FUNCTION "Szukaj_Zmiany" : VOID	// FC 5
//Funkcja wykrywa zmiane w obszarze wejscie i zapamietuje. Umozliwia to wykrycie 
//zmiany stanu kazdego czujnika lini. Funkcja ograniczona jest do dlugosci 32 
//bitow.
//
//Wersja 1.0
//Rozszerzenie dzia³ania funcji do 8 bajtow
AUTHOR : Kng
NAME : Help_FC
VERSION : 0.1
VAR_INPUT
  DWORD_IN_NEW : DWORD ;
END_VAR
VAR_IN_OUT
  DWORD_IN_OLD : DWORD ;
  CHANGE : BOOL ;
END_VAR
VAR_TEMP
  DWORD_TEST : DWORD ;
  Temp_Bit_1 : BOOL ;
  Temp_Bit_2 : BOOL ;
END_VAR
BEGIN
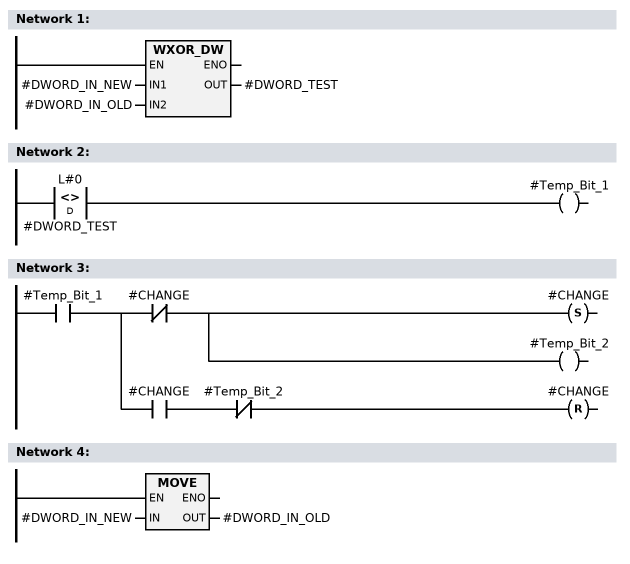
NETWORK
TITLE =
//Sprawdz czy nastapila zmiana
      L     #DWORD_IN_NEW;
      L     #DWORD_IN_OLD;
      XOD;
      T     #DWORD_TEST;
NETWORK
TITLE =
////wykrycie zmiany stanu 
      L     L#0;
      L     #DWORD_TEST;
      <>D;
      =     #Temp_Bit_1;
NETWORK
TITLE =
//Zapisz wykryta zminane
      A     #Temp_Bit_1;
      =     L 5.0;
      A     L 5.0;
      AN    #CHANGE;
      S     #CHANGE;
      =     #Temp_Bit_2;
      A     L 5.0;
      A     #CHANGE;
      AN    #Temp_Bit_2;
      R     #CHANGE;
NETWORK
TITLE =
//Przypisz wartosc obecna jako stara
      L     #DWORD_IN_NEW;
      T     #DWORD_IN_OLD;
END_FUNCTION

FUNCTION "FC_Lampki" : VOID	// FC 6
VERSION : 0.1
VAR_INPUT
  in_0 : BOOL ;
  in_1 : BOOL ;
  in_2 : BOOL ;
  in_3 : BOOL ;
  in_4 : BOOL ;
  in_5 : BOOL ;
  in_6 : BOOL ;
  in_7 : BOOL ;
  Test : BOOL ;
END_VAR
VAR_OUTPUT
  out_0 : BOOL ;
  out_1 : BOOL ;
  out_2 : BOOL ;
  out_3 : BOOL ;
  out_4 : BOOL ;
  out_5 : BOOL ;
  out_6 : BOOL ;
  out_7 : BOOL ;
END_VAR
BEGIN
NETWORK
TITLE =
//przyporzadkowanie wejsc do wyjs
//0
      O     #in_0;
      O     #Test;
      =     #out_0;
//1
      O     #in_1;
      O     #Test;
      =     #out_1;
//2
      O     #in_2;
      O     #Test;
      =     #out_2;
//3
      O     #in_3;
      O     #Test;
      =     #out_3;
//4
      O     #in_4;
      O     #Test;
      =     #out_4;
//5
      O     #in_5;
      O     #Test;
      =     #out_5;
//6
      O     #in_6;
      O     #Test;
      =     #out_6;
//7
      O     #in_7;
      O     #Test;
      =     #out_7;
END_FUNCTION

FUNCTION "Szukaj_Zmiany_2" : VOID	// FC 7
//Funkcja wykrywa zmiane w obszarze wejscie i zapamietuje. Umozliwia to wykrycie 
//zmiany stanu kazdego czujnika lini. Funkcja ograniczona jest do dlugosci 32 
//bitow.
//
//Wersja 1.0
//Rozszerzenie dzia³ania funcji do 8 bajtow
AUTHOR : Kng
NAME : Help_FC
VERSION : 0.1
VAR_INPUT
  DWORD_IN_NEW : DWORD ;
END_VAR
VAR_OUTPUT
  CHANGE : BOOL ;
END_VAR
VAR_IN_OUT
  DWORD_IN_OLD : DWORD ;
END_VAR
BEGIN
NETWORK
TITLE =
//Sprawdz czy nastapila zmiana
      L     #DWORD_IN_NEW;
      L     #DWORD_IN_OLD;
      XOD;
      L     L#0;
      <>D;
      =     #CHANGE;
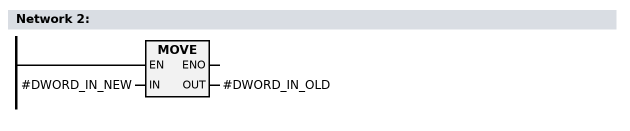
NETWORK
TITLE =
//Przypisz wartosc obecna jako stara
      L     #DWORD_IN_NEW;
      T     #DWORD_IN_OLD;
END_FUNCTION

FUNCTION "Toggle" : VOID	// FC 8
//Funcja zmienia stan wyjscia gdy ktore kolwiek wejscie zostanie wyzwolone
AUTHOR : Kng
NAME : Help_FC
VERSION : 0.1
VAR_INPUT
  Wyzwolenie_1 : BOOL ;
  Wyzwolenie_2 : BOOL ;
  Wyzwolenie_3 : BOOL ;
  Wyzwolenie_4 : BOOL ;
END_VAR
VAR_IN_OUT
  TOGGLE : BOOL ;
END_VAR
VAR_TEMP
  Temp_Bit_2 : BOOL ;
END_VAR
BEGIN
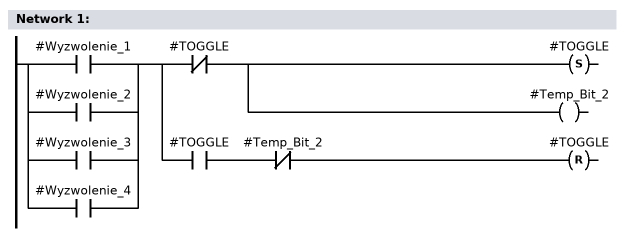
NETWORK
TITLE =
//Zapisz wykryta zminane
      O     #Wyzwolenie_1;
      O     #Wyzwolenie_2;
      O     #Wyzwolenie_3;
      O     #Wyzwolenie_4;
      =     L 1.0;
      A     L 1.0;
      AN    #TOGGLE;
      S     #TOGGLE;
      =     #Temp_Bit_2;
      A     L 1.0;
      A     #TOGGLE;
      AN    #Temp_Bit_2;
      R     #TOGGLE;
END_FUNCTION

FUNCTION "Sterwanie_Swiatlo" : VOID	// FC 9
VERSION : 0.1
VAR_TEMP
  Help_Bit : BOOL ;
END_VAR
BEGIN
NETWORK
TITLE =
//Ten Network celowo jest wolny
NETWORK
TITLE =
//Wyszczegolnienie bledow
//Not AUS Adres 27 (szafa)
//Kod :0001
      A     "Not_Aus_27_OK";
      L     B#16#1;
      JCN   KOD;
//Not AUS Adres 28 (poczatek lini)
//Kod :0010
      A     "Not_Aus_28_OK";
      L     B#16#2;
      JCN   KOD;
//Not AUS Adres 29 (srodek lini)
//Kod :0011
      A     "Not_Aus_29_OK";
      L     B#16#3;
      JCN   KOD;
//Not AUS Adres 30 (koniec lini)
//Kod :0100
      A     "Not_Aus_30_OK";
      L     B#16#4;
      JCN   KOD;
//Sprawdzenie bezpiecznikow w szafie
//Kod:0101
      A     "Fuse_OK";
      L     B#16#5;
      JCN   KOD;
//Sprwadzenie przekaznika bezpieczenstwa
//Kod:0110
      A     "Przekaznik_Bezp_OK";
      L     B#16#6;
      JCN   KOD;
//Sprawdzenie Falownikow Lini    
//Kod:0111
      A     "Falowniki_OK";
      L     B#16#7;
      JCN   KOD;
//Not AUS Adres 31 (koniec lini)
//Kod :1000
      A     "Not_Aus_31_OK";
      L     B#16#8;
      JCN   KOD;
//Sprawdzenie czy jest wlaczony  stop
//Kod:1111
      AN    "Marka_Start_Stop";
      L     B#16#F;
      JCN   KOD;
//Not AUS Adres (Strefa Bindownica)
//Kod :1001
      A     "Strefa_Bind_Zamk";
      L     B#16#9;
      JCN   KOD;
//Not AUS Adres (Strefa Bindownica)
//Kod :1010
      A     "Przek_Rejonu_Bind_Ok";
      L     B#16#10;
      JCN   KOD;
//Brak bledu maszyna pracuje
//Kod:0000
      L     B#16#0;
//Przekaz kod bledu
KOD:  T     "Byte_Bledu";
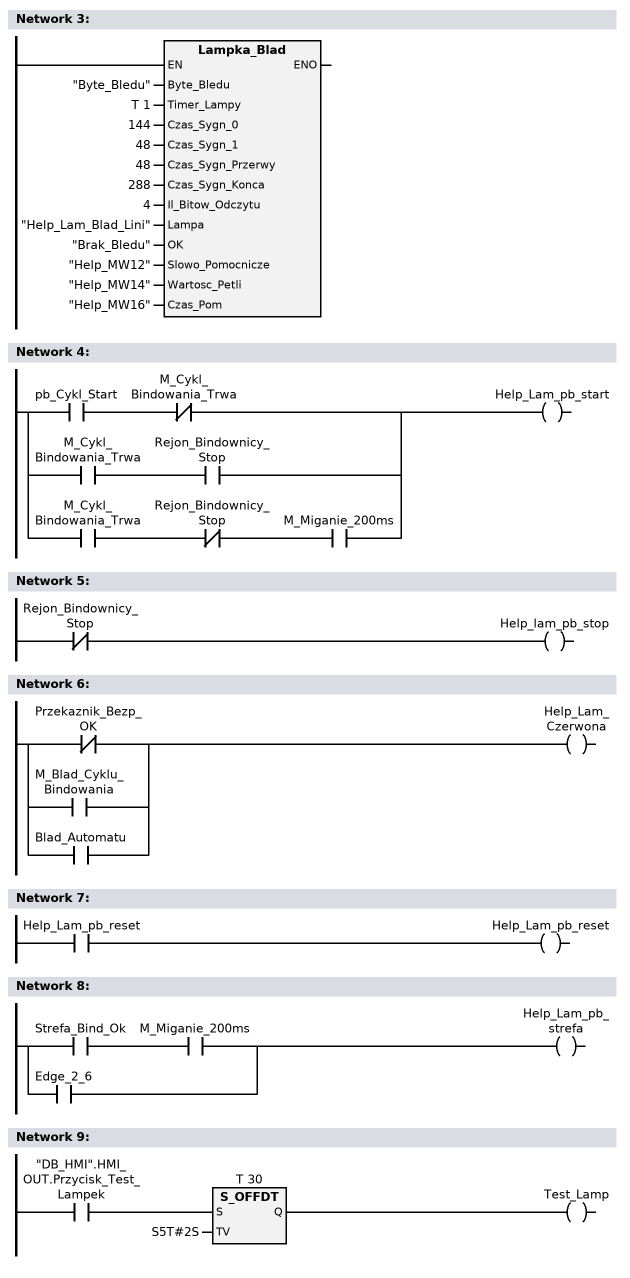
NETWORK
TITLE =
//Lampka bledu
      CALL  "Lampka_Blad" (
           Byte_Bledu               := "Byte_Bledu",
           Timer_Lampy              := T 1,
           Czas_Sygn_0              := 144,
           Czas_Sygn_1              := 48,
           Czas_Sygn_Przerwy        := 48,
           Czas_Sygn_Konca          := 288,
           Il_Bitow_Odczytu         := 4,
           Lampa                    := "Help_Lam_Blad_Lini",
           OK                       := "Brak_Bledu",
           Slowo_Pomocnicze         := "Help_MW12",
           Wartosc_Petli            := "Help_MW14",
           Czas_Pom                 := "Help_MW16");
NETWORK
TITLE =
//Lampka pb start
      A     "pb_Cykl_Start";
      AN    "M_Cykl_Bindowania_Trwa";
      O;
      A     "M_Cykl_Bindowania_Trwa";
      A     "Rejon_Bindownicy_Stop";
      O;
      A     "M_Cykl_Bindowania_Trwa";
      AN    "Rejon_Bindownicy_Stop";
      A     "M_Miganie_200ms";
      =     "Help_Lam_pb_start";
NETWORK
TITLE =
//Lampka stop
      AN    "Rejon_Bindownicy_Stop";
      =     "Help_lam_pb_stop";
NETWORK
TITLE =
      ON    "Przekaznik_Bezp_OK";
      O     "M_Blad_Cyklu_Bindowania";
      O     "Blad_Automatu";
      =     "Help_Lam_Czerwona";
NETWORK
TITLE =
//Miga reset
      A     "Help_Lam_pb_reset";
      =     "Help_Lam_pb_reset";
NETWORK
TITLE =
//Lampka bezpieczenstwa strefa
      A     "Strefa_Bind_Ok";
      A     "M_Miganie_200ms";
      O     "Edge_2_6";
      =     "Help_Lam_pb_strefa";
NETWORK
TITLE =
//Test Lampek z timmerem przedluzonym
      A     "DB_HMI".HMI_OUT.Przycisk_Test_Lampek;
      L     S5T#2S;
      SF    T 30;
      NOP   0;
      NOP   0;
      NOP   0;
      A     T 30;
      =     "Test_Lamp";
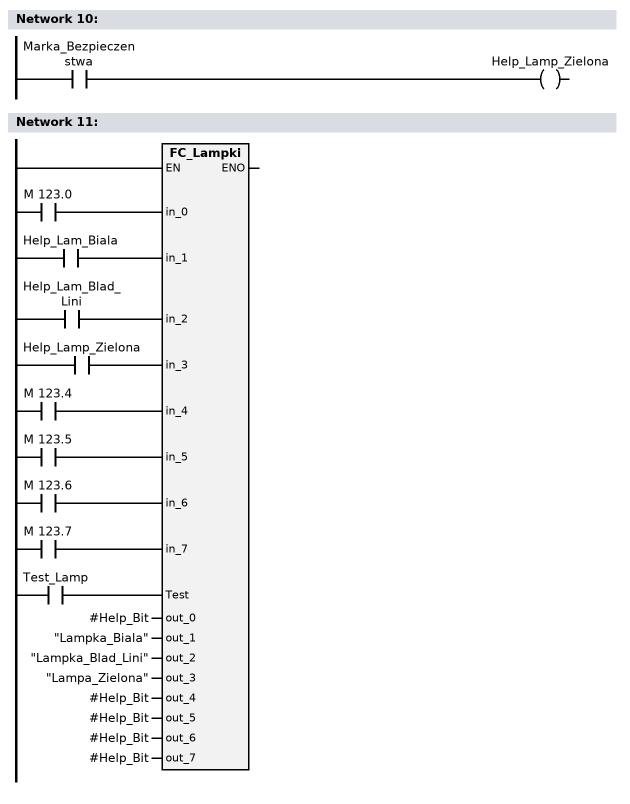
NETWORK
TITLE =
//linia pracuje
      A     "Marka_Bezpieczenstwa";
      =     "Help_Lamp_Zielona";
NETWORK
TITLE =
//Lampki na szafie sterowniczej sa troche przesuniete bo brakuje zielonej
      A     M 123.0;
      =     L 1.0;
      BLD   103;
      A     "Help_Lam_Biala";
      =     L 1.1;
      BLD   103;
      A     "Help_Lam_Blad_Lini";
      =     L 1.2;
      BLD   103;
      A     "Help_Lamp_Zielona";
      =     L 1.3;
      BLD   103;
      A     M 123.4;
      =     L 1.4;
      BLD   103;
      A     M 123.5;
      =     L 1.5;
      BLD   103;
      A     M 123.6;
      =     L 1.6;
      BLD   103;
      A     M 123.7;
      =     L 1.7;
      BLD   103;
      A     "Test_Lamp";
      =     L 2.0;
      BLD   103;
      CALL  "FC_Lampki" (
           in_0                     := L 1.0,
           in_1                     := L 1.1,
           in_2                     := L 1.2,
           in_3                     := L 1.3,
           in_4                     := L 1.4,
           in_5                     := L 1.5,
           in_6                     := L 1.6,
           in_7                     := L 1.7,
           Test                     := L 2.0,
           out_0                    := #Help_Bit,
           out_1                    := "Lampka_Biala",
           out_2                    := "Lampka_Blad_Lini",
           out_3                    := "Lampa_Zielona",
           out_4                    := #Help_Bit,
           out_5                    := #Help_Bit,
           out_6                    := #Help_Bit,
           out_7                    := #Help_Bit);
      NOP   0;
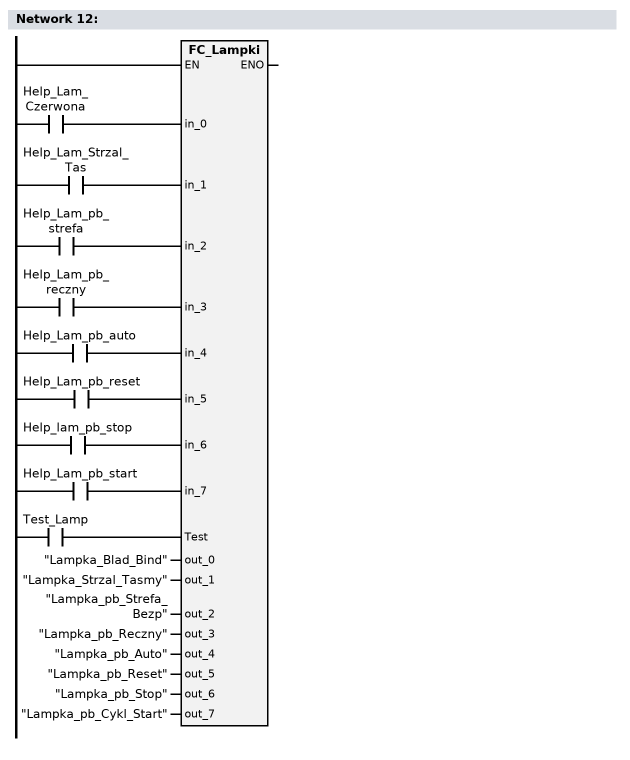
NETWORK
TITLE =
//funkcja zarzadzajaca lampami
//Lampki na panelu operatorskim
      A     "Help_Lam_Czerwona";
      =     L 1.0;
      BLD   103;
      A     "Help_Lam_Strzal_Tas";
      =     L 1.1;
      BLD   103;
      A     "Help_Lam_pb_strefa";
      =     L 1.2;
      BLD   103;
      A     "Help_Lam_pb_reczny";
      =     L 1.3;
      BLD   103;
      A     "Help_Lam_pb_auto";
      =     L 1.4;
      BLD   103;
      A     "Help_Lam_pb_reset";
      =     L 1.5;
      BLD   103;
      A     "Help_lam_pb_stop";
      =     L 1.6;
      BLD   103;
      A     "Help_Lam_pb_start";
      =     L 1.7;
      BLD   103;
      A     "Test_Lamp";
      =     L 2.0;
      BLD   103;
      CALL  "FC_Lampki" (
           in_0                     := L 1.0,
           in_1                     := L 1.1,
           in_2                     := L 1.2,
           in_3                     := L 1.3,
           in_4                     := L 1.4,
           in_5                     := L 1.5,
           in_6                     := L 1.6,
           in_7                     := L 1.7,
           Test                     := L 2.0,
           out_0                    := "Lampka_Blad_Bind",
           out_1                    := "Lampka_Strzal_Tasmy",
           out_2                    := "Lampka_pb_Strefa_Bezp",
           out_3                    := "Lampka_pb_Reczny",
           out_4                    := "Lampka_pb_Auto",
           out_5                    := "Lampka_pb_Reset",
           out_6                    := "Lampka_pb_Stop",
           out_7                    := "Lampka_pb_Cykl_Start");
      NOP   0;
END_FUNCTION

FUNCTION "Lampka_Blad" : VOID	// FC 10
//Funkcja odowiada za generowanie kodu bledu w postaci sekwencji impulsow 
//swietlnych. Maksymalna ilosc imulsow kodu wynosi 8(dl. jednego bajtu).
//Przyukladowa sekwencja kodu to 0001 (sygnal: krotki,krotki,krotki,dlugi).
//
//Kod braku bledu to 0000-przy ustawionej liczbie bitow odczytywanych na 4
//
AUTHOR : Kng
NAME : Error
VERSION : 0.1
VAR_INPUT
  Byte_Bledu : BYTE ;	//Byte wejsciowy kodu bledu
  Timer_Lampy : TIMER ;
  Czas_Sygn_0 : S5TIME ;	//Czas sygnalu dla zera
  Czas_Sygn_1 : S5TIME ;	//Czas sygnalu dla jeden
  Czas_Sygn_Przerwy : S5TIME ;	//Czas sygnalu przerwy pomiedzy impulsami
  Czas_Sygn_Konca : S5TIME ;	//Czas sygnalu konca sekwencji bledu
  Il_Bitow_Odczytu : INT ;	//Ilosc bitow odczytu sekwencji
END_VAR
VAR_OUTPUT
  Lampa : BOOL ;	//Wyjscie sterujace lampa
  OK : BOOL ;	//Brak bledow kod:0000
END_VAR
VAR_IN_OUT
  Slowo_Pomocnicze : WORD ;	//Slowo pomocnicze
  Wartosc_Petli : INT ;	//Wartosc petli
  Czas_Pom : S5TIME ;
END_VAR
VAR_TEMP
  Help_Edge_1 : BOOL ;
  Help_Edge_2 : BOOL ;
  Help_Edge_3 : BOOL ;
  Help_Edge_4 : BOOL ;
  Help_Edge_5 : BOOL ;
  Help_Lampa : BOOL ;
  Help_Timer_Gora : BOOL ;
  Help_Przerwa : BOOL ;
  Help_Timer_Dol : BOOL ;
  Help_Sek_Kon : BOOL ;
  Help_Timer_Kon : BOOL ;
  Help_Powrot : BOOL ;
  Help_Bit_Stop : BOOL ;
  Help_Bit_1_5 : BOOL ;
  Help_Bit_1_6 : BOOL ;
  Help_Bit_1_7 : BOOL ;
  Help_Word_2 : WORD ;
END_VAR
BEGIN
NETWORK
TITLE =
//Funkcja nie wykrywa bledu gdy transmisja 0000
      L     #Byte_Bledu;
      L     0;
      ==I;
      R     #Help_Bit_Stop;
      JC    good;
      L     #Byte_Bledu;
      L     B#16#F;
      ==I;
      JC    stop;
// Odczytanie zmiennych pomocniczych
      L     #Slowo_Pomocnicze;
      T     LW 0;
//Wyznaczenie sekwencji bledu
NETWORK
TITLE =
      O     #Help_Timer_Gora;
      O     #Help_Timer_Dol;
      O     #Help_Timer_Kon;
      JC    play;
// Sekwencja konca
      A     #Help_Sek_Kon;
      JCN   et_4;
      SET;
      S     #Help_Timer_Kon;
      L     #Czas_Sygn_Konca;
      T     #Czas_Pom;
      JU    play;
et_4: NOP   0;
//Sekwencja przerwy
      A     #Help_Przerwa;
      JCN   et_1;
      SET;
      S     #Help_Timer_Dol;
      L     #Czas_Sygn_Przerwy;
      T     #Czas_Pom;
      JU    play;
et_1: NOP   0;
//Wyznaczenie sekwencji bledu
//     L     #Il_Bitow_Odczytu           //skres to by uzyskac czytanie w druga
      L     #Wartosc_Petli;
      L     1;
      -I;
      L     #Byte_Bledu;
      SRW;
      T     #Help_Word_2;
//Zabranie bitu sekwencji
      A     L 3.0;	//bit po przesunieciu o odpowiednia sekwencje
      JCN   et_0;
//Czas sygnalu krotkiego
      SET;
      =     #Help_Timer_Gora;
      L     #Czas_Sygn_1;
      T     #Czas_Pom;
      JU    play;
et_0: NOP   0;
//Czas sygnalu dlugiego
      SET;
      =     #Help_Timer_Gora;
      L     #Czas_Sygn_0;
      T     #Czas_Pom;
      JU    play;
//Puszczenie sygnalu timer'a
//***************************************************************
play: O     #Help_Timer_Gora;
      O     #Help_Timer_Dol;
      O     #Help_Timer_Kon;
      AN    #Help_Powrot;
      L     #Czas_Pom;
      SE    #Timer_Lampy;
      A     #Timer_Lampy;
      =     #Help_Lampa;
//***************************************************************
//Przejscie do przerwy
      A     #Help_Timer_Gora;
      A     #Help_Lampa;
      FN    #Help_Edge_2;
      S     #Help_Przerwa;
      R     #Help_Edge_2;
      R     #Help_Timer_Gora;
      JC    play;
//Reset przerwy
      A     #Help_Timer_Dol;
      A     #Help_Lampa;
      FN    #Help_Edge_3;
      R     #Help_Przerwa;
      R     #Help_Edge_3;
      R     #Help_Timer_Dol;
      JC    play;
//Uruchomienie timer'a konca sekwencji
      A     #Help_Timer_Kon;
      A     #Help_Lampa;
      FN    #Help_Edge_5;
      R     #Help_Sek_Kon;
      R     #Help_Timer_Kon;
      R     #Help_Edge_5;
      JC    play;
//Dekrementacja licznika przesuniec bitow
      A     #Help_Przerwa;
      FP    #Help_Edge_4;
      JCN   et_2;
      L     #Wartosc_Petli;
      L     1;
      -I;
      T     #Wartosc_Petli;
et_2: NOP   0;
//Sekwencja konczaca
      L     #Wartosc_Petli;
      L     0;
      <=I;
      JCN   et_3;
      SET;
      S     #Help_Sek_Kon;
      L     #Il_Bitow_Odczytu;
      T     #Wartosc_Petli;
et_3: NOP   0;
NETWORK
TITLE =
//Wystawienie wyjsc
      A     #Help_Timer_Gora;
      A     #Help_Lampa;
      AN    #Help_Timer_Dol;
      AN    #Help_Timer_Kon;
      =     #Lampa;
NETWORK
TITLE =
      SET;
      R     #Help_Powrot;
      R     #OK;
      L     LW 0;
      T     #Slowo_Pomocnicze;
      BEU;
NETWORK
TITLE =
stop: NOP   0;
      SET;
      S     #Help_Bit_Stop;
good: NOP   0;
      A     #Help_Bit_Stop;
      =     #Lampa;
//wyzeruj wartosci pomocnicze
      L     0;
      T     LW 0;
//Przypisz ilosc petli by zaczynac od pelnego bledu
      L     #Il_Bitow_Odczytu;
      T     #Wartosc_Petli;
//Wylaczenie swiecenie lampy  i umozliwienie powrotu do pracujacego timera
      SET;
      R     #Help_Bit_Stop;
      R     #Timer_Lampy;
      S     #Help_Powrot;
      S     #OK;
      L     LW 0;
      T     #Slowo_Pomocnicze;
END_FUNCTION

FUNCTION "Przyporzadkowanie_Wejsc" : VOID	// FC 20
//Pobranie z bloku db stanu wejsc sieci asi i przyporzadkowanie do odpowiedniego 
//urzadzenia lini.
//NW35-adresy B
//
//
//Opis sygnalow od bindownicy:
//banda 23, 24, 1, 2 tworza zestaw tasm maszyny bindujacej
//obr 15 to obrotnica bindownicy
//25,26- to kurtyny
//16-rygiel
//17-modul resetu
AUTHOR : Kng
NAME : Help_FC
VERSION : 0.1
VAR_TEMP
  Help_Bit_1 : BOOL ;
  Help_Bit_2 : BOOL ;
  Help_Word_1 : INT ;
  Help_Word_2 : INT ;
END_VAR
BEGIN
NETWORK
TITLE =
//Ten network celowo jest wolny
NETWORK
TITLE =
NETWORK
TITLE = Silnik ok
//Banda Adres 1
      A     "Asi_input".Adres_1_bit_0;
      O     "Zawsze_True";	//dodane
      =     "AIO".Banda_1.Silnik_OK;
      A     "Asi_input".Adres_1_bit_1;
      =     "AIO".Banda_1.Rezerwa_Silnik;
      A     "Asi_input".Adres_1_bit_2;
      =     "AIO".Banda_1.Foto_1;
      A     "Asi_input".Adres_1_bit_3;
      =     "AIO".Banda_1.Foto_2;
NETWORK
TITLE = Silnik ok
//Banda Adres 2
      A     "Asi_input".Adres_2_bit_0;
      O     "Zawsze_True";
      =     "AIO".Banda_2.Silnik_OK;
      A     "Asi_input".Adres_2_bit_1;
      =     "AIO".Banda_2.Rezerwa_Silnik;
      A     "Asi_input".Adres_2_bit_2;
      =     "AIO".Banda_2.Foto_1;
      A     "Asi_input".Adres_2_bit_3;
      =     "AIO".Banda_2.Foto_2;
NETWORK
TITLE = Silnik ok
//Banda Adres 3
      A     "Asi_input".Adres_3_bit_0;
      =     "AIO".Banda_3.Silnik_OK;
      A     "Asi_input".Adres_3_bit_1;
      =     "AIO".Banda_3.Rezerwa_Silnik;
      A     "Asi_input".Adres_3_bit_2;
      =     "AIO".Banda_3.Foto_1;
      A     "Asi_input".Adres_3_bit_3;
      =     "AIO".Banda_3.Foto_2;
NETWORK
TITLE = Silnik ok
//Banda Adres 4
      A     "Asi_input".Adres_4_bit_0;
      =     "AIO".Banda_4.Silnik_OK;
      A     "Asi_input".Adres_4_bit_1;
      =     "AIO".Banda_4.Rezerwa_Silnik;
      A     "Asi_input".Adres_4_bit_2;
      =     "AIO".Banda_4.Foto_1;
      A     "Asi_input".Adres_4_bit_3;
      =     "AIO".Banda_4.Foto_2;
NETWORK
TITLE = Silnik ok
//Banda Adres 5
      A     "Asi_input".Adres_5_bit_0;
      =     "AIO".Banda_5.Silnik_OK;
      A     "Asi_input".Adres_5_bit_1;
      =     "AIO".Banda_5.Rezerwa_Silnik;
      A     "Asi_input".Adres_5_bit_2;
      =     "AIO".Banda_5.Foto_1;
      A     "Asi_input".Adres_5_bit_3;
      =     "AIO".Banda_5.Foto_2;
NETWORK
TITLE = Silnik ok
//Banda Adres 6
      A     "Asi_input".Adres_6_bit_0;
      =     "AIO".Banda_6.Silnik_OK;
      A     "Asi_input".Adres_6_bit_1;
      =     "AIO".Banda_6.Rezerwa_Silnik;
      A     "Asi_input".Adres_6_bit_2;
      =     "AIO".Banda_6.Foto_1;
      A     "Asi_input".Adres_6_bit_3;
      =     "AIO".Banda_6.Foto_2;
NETWORK
TITLE = Silnik ok
//Banda Adres 7
      A     "Asi_input".Adres_7_bit_0;
      =     "AIO".Banda_7.Silnik_OK;
      A     "Asi_input".Adres_7_bit_1;
      =     "AIO".Banda_7.Rezerwa_Silnik;
      A     "Asi_input".Adres_7_bit_2;
      =     "AIO".Banda_7.Foto_1;
      A     "Asi_input".Adres_7_bit_3;
      =     "AIO".Banda_7.Foto_2;
NETWORK
TITLE = Silnik ok
//Banda Adres 8
      A     "Asi_input".Adres_8_bit_0;
      =     "AIO".Banda_8.Silnik_OK;
      A     "Asi_input".Adres_8_bit_1;
      =     "AIO".Banda_8.Rezerwa_Silnik;
      A     "Asi_input".Adres_8_bit_2;
      =     "AIO".Banda_8.Foto_1;
      A     "Asi_input".Adres_8_bit_3;
      =     "AIO".Banda_8.Foto_2;
NETWORK
TITLE = Silnik ok
//Banda Adres 9
      A     "Asi_input".Adres_9_bit_0;
      =     "AIO".Banda_9.Silnik_OK;
      A     "Asi_input".Adres_9_bit_1;
      =     "AIO".Banda_9.Rezerwa_Silnik;
      A     "Asi_input".Adres_9_bit_2;
      =     "AIO".Banda_9.Foto_1;
      A     "Asi_input".Adres_9_bit_3;
      =     "AIO".Banda_9.Foto_2;
//Info do foliarki o zajetosci lini
      A     "AIO".Banda_9.Foto_1;
      =     "MPI_GD".OUT.Foto_Banda_9;
//-
NETWORK
TITLE = Silnik ok
//Banda Adres 10.Banda nalezy do foliarki.
      A     "Asi_input".Adres_10_bit_0;
      =     "AIO".Banda_10.Silnik_OK;
      A     "Asi_input".Adres_10_bit_1;
      =     "AIO".Banda_10.Rezerwa_Silnik;
      A     "Asi_input".Adres_10_bit_2;
      =     "AIO".Banda_10.Foto_1;
      A     "Asi_input".Adres_10_bit_3;
      =     "AIO".Banda_10.Foto_2;
//Sygnaly do foliarki
      A     "AIO".Banda_10.Silnik_OK;
      =     "MPI_GD".OUT.Silnik_10_OK;
//-
      A     "AIO".Banda_10.Foto_1;
      =     "MPI_GD".OUT.Foto_1_Banda_10;
//-
      A     "AIO".Banda_10.Foto_2;
      =     "MPI_GD".OUT.Foto_2_Banda_10;
NETWORK
TITLE = Silnik ok
//Banda Adres 11. Banda nalezy do foliarki.
      A     "Asi_input".Adres_11_bit_0;
      =     "AIO".Banda_11.Silnik_OK;
      A     "Asi_input".Adres_11_bit_1;
      =     "AIO".Banda_11.Rezerwa_Silnik;
      A     "Asi_input".Adres_11_bit_2;
      =     "AIO".Banda_11.Foto_1;
      A     "Asi_input".Adres_11_bit_3;
      =     "AIO".Banda_11.Foto_2;
//Sygnaly do foliarki
      A     "AIO".Banda_11.Silnik_OK;
      =     "MPI_GD".OUT.Silnik_11_OK;
//-
      A     "AIO".Banda_11.Foto_1;
      =     "MPI_GD".OUT.Foto_Banda_11;
NETWORK
TITLE = Silnik ok
//Banda Adres 12
      A     "Asi_input".Adres_12_bit_0;
      =     "AIO".Banda_12.Silnik_OK;
      A     "Asi_input".Adres_12_bit_1;
      =     "AIO".Banda_12.Rezerwa_Silnik;
      A     "Asi_input".Adres_12_bit_2;
      =     "AIO".Banda_12.Foto_1;
      A     "Asi_input".Adres_12_bit_3;
      =     "AIO".Banda_12.Foto_2;
NETWORK
TITLE = Silnik ok
//Banda Adres 13
      A     "Asi_input".Adres_13_bit_0;
      =     "AIO".Banda_13.Silnik_OK;
      A     "Asi_input".Adres_13_bit_1;
      =     "AIO".Banda_13.Rezerwa_Silnik;
      A     "Asi_input".Adres_13_bit_2;
      =     "AIO".Banda_13.Foto_1;
      A     "Asi_input".Adres_13_bit_3;
      =     "AIO".Banda_13.Foto_2;
NETWORK
TITLE = Silnik ok
//Banda Adres 14
      A     "Asi_input".Adres_14_bit_0;
      =     "AIO".Banda_14.Silnik_OK;
      A     "Asi_input".Adres_14_bit_1;
      =     "AIO".Banda_14.Rezerwa_Silnik;
      A     "Asi_input".Adres_14_bit_2;
      =     "AIO".Banda_14.Foto_1;
      A     "Asi_input".Adres_14_bit_3;
      =     "AIO".Banda_14.Foto_2;
NETWORK
TITLE = Silnik ok
//Obrotnica Adres 15
      A     "Asi_input".Adres_15_bit_0;
      =     "AIO".Obr_15.Silnik_OK;
      A     "Asi_input".Adres_15_bit_1;
      =     "AIO".Obr_15.Rezerwa_Silnik;
      A     "Asi_input".Adres_15_bit_2;
      =     "AIO".Obr_15.Foto_1;
      A     "Asi_input".Adres_15_bit_3;
      =     "AIO".Obr_15.Foto_2;
NETWORK
TITLE = Silnik ok
//Uwaga modul safety !!!
//Rygiel Adres 16
      A     "Asi_input".Adres_16_bit_0;
      =     "AIO".Rygiel_16.OSSD_Tor_1_1;
      A     "Asi_input".Adres_16_bit_1;
      =     "AIO".Rygiel_16.OSSD_Tor_1_2;
      A     "Asi_input".Adres_16_bit_2;
      =     "AIO".Rygiel_16.OSSD_Tor_2_1;
      A     "Asi_input".Adres_16_bit_3;
      =     "AIO".Rygiel_16.OSSD_Tor_2_2;
NETWORK
TITLE = Silnik ok
//Reset kurtyn bezpieczenswa Adres 17
//Nie wykorzystywane wejscia
NETWORK
TITLE = Silnik ok
//Obrotnica Adres_18
      A     "Asi_input".Adres_18_bit_0;
      =     "AIO".Obr_18.Silnik_OK;
      A     "Asi_input".Adres_18_bit_1;
      =     "AIO".Obr_18.Rezerwa_Silnik;
      A     "Asi_input".Adres_18_bit_2;
      =     "AIO".Obr_18.Foto_1;
      A     "Asi_input".Adres_18_bit_3;
      =     "AIO".Obr_18.Foto_2;
NETWORK
TITLE = Silnik ok
//Czujniki obrotnicy 1 Adres 19
      A     "Asi_input".Adres_19_bit_0;
      =     "AIO".Czuj_19.Czujnik_0_St;
      A     "Asi_input".Adres_19_bit_1;
      =     "AIO".Czuj_19.Czujnik_Ham_0_St;
      A     "Asi_input".Adres_19_bit_2;
      =     "AIO".Czuj_19.Czujnik_Ham_90_St;
      A     "Asi_input".Adres_19_bit_3;
      =     "AIO".Czuj_19.Czujnik_90_St;
NETWORK
TITLE = Silnik ok
//Obrotnica Adres 20
      A     "Asi_input".Adres_20_bit_0;
      =     "AIO".Obr_20.Silnik_OK;
      A     "Asi_input".Adres_20_bit_1;
      =     "AIO".Obr_20.Rezerwa_Silnik;
      A     "Asi_input".Adres_20_bit_2;
      =     "AIO".Obr_20.Foto_1;
      A     "Asi_input".Adres_20_bit_3;
      =     "AIO".Obr_20.Foto_2;
NETWORK
TITLE = Silnik ok
//Czujniki Obrotnicy 2 Adres 21
      A     "Asi_input".Adres_21_bit_0;
      =     "AIO".Czuj_21.Czujnik_0_St;
      A     "Asi_input".Adres_21_bit_1;
      =     "AIO".Czuj_21.Czujnik_Ham_0_St;
      A     "Asi_input".Adres_21_bit_2;
      =     "AIO".Czuj_21.Czujnik_Ham_90_St;
      A     "Asi_input".Adres_21_bit_3;
      =     "AIO".Czuj_21.Czujnik_90_St;
NETWORK
TITLE = Silnik ok
//Czujniki Obrotnicy 2 Adres 22
      A     "Asi_input".Adres_22_bit_0;
      =     "AIO".Czuj_22.Czujnik_45_St_CW;
      A     "Asi_input".Adres_22_bit_1;
      =     "AIO".Czuj_22.Czujnik_45_St_CCW;
      A     "Asi_input".Adres_22_bit_2;
      =     "AIO".Czuj_22.Rez_0_2;
      A     "Asi_input".Adres_22_bit_3;
      =     "AIO".Czuj_22.Rez_0_3;
NETWORK
TITLE = Wejscie SEW 1
//Banda 23 znajdujaca sie bedaca banda wjazdowa do bindownicy
      A     "Asi_input".Adres_23_bit_0;
      =     "AIO".Banda_23.Silnik_OK;
      A     "Asi_input".Adres_23_bit_1;
      =     "AIO".Banda_23.Rezerwa_Silnik;
      A     "Asi_input".Adres_23_bit_2;
      =     "AIO".Banda_23.Foto_1;
      A     "Asi_input".Adres_23_bit_3;
      =     "AIO".Banda_23.Foto_2;
NETWORK
TITLE = Silnik ok
//Banda 24
      A     "Asi_input".Adres_24_bit_0;
      =     "AIO".Banda_24.Silnik_OK;
      A     "Asi_input".Adres_24_bit_1;
      =     "AIO".Banda_24.Rezerwa_Silnik;
      A     "Asi_input".Adres_24_bit_2;
      =     "AIO".Banda_24.Foto_1;
      A     "Asi_input".Adres_24_bit_3;
      =     "AIO".Banda_24.Foto_2;
NETWORK
TITLE =
//Sprawdzenie czujnikow Bezpieczenstwa lini
//Kurtyna 25
      A     "Asi_input".Adres_25_bit_0;
      =     "AIO".Kurtyna_25.OSSD_Tor_1_1;
      A     "Asi_input".Adres_25_bit_1;
      =     "AIO".Kurtyna_25.OSSD_Tor_1_2;
      A     "Asi_input".Adres_25_bit_2;
      =     "AIO".Kurtyna_25.OSSD_Tor_2_1;
      A     "Asi_input".Adres_25_bit_3;
      =     "AIO".Kurtyna_25.OSSD_Tor_2_2;
NETWORK
TITLE =
//Sprawdzenie czujnikow Bezpieczenstwa lini
//Kurtyna 26
      A     "Asi_input".Adres_26_bit_0;
      =     "AIO".Kurtyna_26.OSSD_Tor_1_1;
      A     "Asi_input".Adres_26_bit_1;
      =     "AIO".Kurtyna_26.OSSD_Tor_1_2;
      A     "Asi_input".Adres_26_bit_2;
      =     "AIO".Kurtyna_26.OSSD_Tor_2_1;
      A     "Asi_input".Adres_26_bit_3;
      =     "AIO".Kurtyna_26.OSSD_Tor_2_2;
NETWORK
TITLE = Silnik ok
//Sprawdzenie czujnikow Bezpieczenstwa lini
//Not Aus 27
      A     "Asi_input".Adres_27_bit_0;
      =     "AIO".ESTOP_27.EStop_Tor_1_1;
      A     "Asi_input".Adres_27_bit_1;
      =     "AIO".ESTOP_27.EStop_Tor_1_2;
      A     "Asi_input".Adres_27_bit_2;
      =     "AIO".ESTOP_27.EStop_Tor_2_1;
      A     "Asi_input".Adres_27_bit_3;
      =     "AIO".ESTOP_27.EStop_Tor_2_2;
NETWORK
TITLE =
//Sprawdzenie czujnikow Bezpieczenstwa lini
//Not Aus 28
      A     "Asi_input".Adres_28_bit_0;
      =     "AIO".ESTOP_28.EStop_Tor_1_1;
      A     "Asi_input".Adres_28_bit_1;
      =     "AIO".ESTOP_28.EStop_Tor_1_2;
      A     "Asi_input".Adres_28_bit_2;
      =     "AIO".ESTOP_28.EStop_Tor_2_1;
      A     "Asi_input".Adres_28_bit_3;
      =     "AIO".ESTOP_28.EStop_Tor_2_2;
NETWORK
TITLE =
//Sprawdzenie czujnikow Bezpieczenstwa lini
//Not Aus 29
      A     "Asi_input".Adres_29_bit_0;
      =     "AIO".ESTOP_29.EStop_Tor_1_1;
      A     "Asi_input".Adres_29_bit_1;
      =     "AIO".ESTOP_29.EStop_Tor_1_2;
      A     "Asi_input".Adres_29_bit_2;
      =     "AIO".ESTOP_29.EStop_Tor_2_1;
      A     "Asi_input".Adres_29_bit_3;
      =     "AIO".ESTOP_29.EStop_Tor_2_2;
NETWORK
TITLE =
//Sprawdzenie czujnikow Bezpieczenstwa lini
//Not Aus 30
      A     "Asi_input".Adres_30_bit_0;
      =     "AIO".ESTOP_30.EStop_Tor_1_1;
      A     "Asi_input".Adres_30_bit_1;
      =     "AIO".ESTOP_30.EStop_Tor_1_2;
      A     "Asi_input".Adres_30_bit_2;
      =     "AIO".ESTOP_30.EStop_Tor_2_1;
      A     "Asi_input".Adres_30_bit_3;
      =     "AIO".ESTOP_30.EStop_Tor_2_2;
NETWORK
TITLE =
//Sprawdzenie czujnikow Bezpieczenstwa lini
//Not Aus 31
      A     "Asi_input".Adres_31_bit_0;
      =     "AIO".ESTOP_31.EStop_Tor_1_1;
      A     "Asi_input".Adres_31_bit_1;
      =     "AIO".ESTOP_31.EStop_Tor_1_2;
      A     "Asi_input".Adres_31_bit_2;
      =     "AIO".ESTOP_31.EStop_Tor_2_1;
      A     "Asi_input".Adres_31_bit_3;
      =     "AIO".ESTOP_31.EStop_Tor_2_2;
NETWORK
TITLE =
//Segment adresow B
//Dotyczy jedynie bialych modulow inuput nie zawartych wyzej
NETWORK
TITLE =
//Czujnik bindownicy Adres 19B 
      A     "Asi_input".B_Adres_19_bit_0;
      =     "AIO".Czuj_19_B.Czujnik_0_St;
      A     "Asi_input".B_Adres_19_bit_1;
      =     "AIO".Czuj_19_B.Czujnik_Ham_0_St;
      A     "Asi_input".B_Adres_19_bit_2;
      =     "AIO".Czuj_19_B.Czujnik_Ham_90_St;
      A     "Asi_input".B_Adres_19_bit_3;
      =     "AIO".Czuj_19_B.Czujnik_90_St;
NETWORK
TITLE =
//Czujnik bindownicy Adres 17B 
      A     "Asi_input".B_Adres_17_bit_0;
      =     "AIO".Czuj_17_B.Czujnik_Ham_180_St;
      A     "Asi_input".B_Adres_17_bit_1;
      =     "AIO".Czuj_17_B.Czujnik_180_St;
      A     "Asi_input".B_Adres_17_bit_2;
      =     "AIO".Czuj_17_B.Czujnik_Ham_270_St;
      A     "Asi_input".B_Adres_17_bit_3;
      =     "AIO".Czuj_17_B.Czujnik_270_St;
END_FUNCTION

FUNCTION "Przyporzadkowanie_Wyjsc" : VOID	// FC 21
VERSION : 0.1
VAR_TEMP
  Temp_Word_1 : INT ;
  Help_Bit_1 : BOOL ;
END_VAR
BEGIN
NETWORK
TITLE =
//Ten Network celowo jest wolny
NETWORK
TITLE = Temporary placeholder variable
//Banda 1 Adres 1
//****************ClockWise*******************
      A     "AIO".Banda_1.CC_Wise;	//C_Wise
      =     "Asi_output".Adres_1_bit_0;
//****************CounterClockWise************
      A     "AIO".Banda_1.C_Wise;
      =     "Asi_output".Adres_1_bit_1;	//CC_Wise
//****************Wolno***********************
      A     "AIO".Banda_1.Wolno;
      O     "pb_Strefa_bezpieczenstwa";
      =     "Asi_output".Adres_1_bit_2;	//Wolno
//****************Bit_Bezpieczenstwa**********
      A     "Marka_Bezpieczenstwa";	//Safety
      =     "Asi_output".Adres_1_bit_3;
NETWORK
TITLE = Temporary placeholder variable
//Banda 2 Adres 2
//****************ClockWise*******************
      A     "AIO".Banda_2.CC_Wise;	//C_Wise
      =     "Asi_output".Adres_2_bit_0;
//****************CounterClockWise************
      A     "AIO".Banda_2.C_Wise;
      =     "Asi_output".Adres_2_bit_1;	//CC_Wise
//****************Wolno***********************
      AN    "AIO".Banda_2.Wolno;
      =     "Asi_output".Adres_2_bit_2;	//Wolno
//****************Bit_Bezpieczenstwa**********
      A     "Marka_Bezpieczenstwa";	//Safety
      =     "Asi_output".Adres_2_bit_3;
NETWORK
TITLE = Temporary placeholder variable
//Banda 3 Adres 3
//****************ClockWise*******************
      A     "Zawsze_False";	//C_Wise
      =     "Asi_output".Adres_3_bit_0;
//****************CounterClockWise************
      A     "AIO".Banda_3.C_Wise;
      =     "Asi_output".Adres_3_bit_1;	//CC_Wise
//****************Wolno***********************
      A     "Zawsze_True";
      =     "Asi_output".Adres_3_bit_2;	//Wolno
//****************Bit_Bezpieczenstwa**********
      A     "Marka_Bezpieczenstwa";	//Safety
      =     "Asi_output".Adres_3_bit_3;
NETWORK
TITLE = Temporary placeholder variable
//Banda 4 Obrotnica
//****************ClockWise*******************
      A     "AIO".Banda_4.C_Wise;	//C_Wise
      =     "Asi_output".Adres_4_bit_0;
//****************CounterClockWise************
      A     "AIO".Banda_4.CC_Wise;
      =     "Asi_output".Adres_4_bit_1;	//CC_Wise
//****************Wolno***********************
      A     "Zawsze_True";
      =     "Asi_output".Adres_4_bit_2;	//Wolno
//****************Bit_Bezpieczenstwa**********
      A     "Marka_Bezpieczenstwa";	//Safety
      =     "Asi_output".Adres_4_bit_3;
NETWORK
TITLE = Temporary placeholder variable
//Banda 5 Rolki
//****************ClockWise*******************
      A     "Zawsze_False";	//C_Wise
      =     "Asi_output".Adres_5_bit_0;
//****************CounterClockWise************
      A     "AIO".Banda_5.C_Wise;
      =     "Asi_output".Adres_5_bit_1;	//CC_Wise
//****************Wolno***********************
      A     "Zawsze_True";
      =     "Asi_output".Adres_5_bit_2;	//Wolno
//****************Bit_Bezpieczenstwa**********
      A     "Marka_Bezpieczenstwa";	//Safety
      =     "Asi_output".Adres_5_bit_3;
NETWORK
TITLE = Temporary placeholder variable
//Banda 6 Rolki
//****************ClockWise*******************
      A     "AIO".Banda_6.C_Wise;	//C_Wise
      =     "Asi_output".Adres_6_bit_0;
//****************CounterClockWise************
      A     "Zawsze_False";
      =     "Asi_output".Adres_6_bit_1;	//CC_Wise
//****************Wolno***********************
      A     "Zawsze_False";
      =     "Asi_output".Adres_6_bit_2;	//Wolno
//****************Bit_Bezpieczenstwa**********
      A     "Marka_Bezpieczenstwa";	//Safety
      =     "Asi_output".Adres_6_bit_3;
NETWORK
TITLE = Temporary placeholder variable
//Banda 7 Rolki
//****************ClockWise*******************
      A     "Zawsze_False";	//C_Wise
      =     "Asi_output".Adres_7_bit_0;
//****************CounterClockWise************
      A     "AIO".Banda_7.C_Wise;
      =     "Asi_output".Adres_7_bit_1;	//CC_Wise
//****************Wolno***********************
      A     "Zawsze_True";
      =     "Asi_output".Adres_7_bit_2;	//Wolno
//****************Bit_Bezpieczenstwa**********
      A     "Marka_Bezpieczenstwa";	//Safety
      =     "Asi_output".Adres_7_bit_3;
NETWORK
TITLE = Temporary placeholder variable
//Banda 8 Rolki
//****************ClockWise*******************
      A     "AIO".Banda_8.C_Wise;	//C_Wise
      =     "Asi_output".Adres_8_bit_0;
//****************CounterClockWise************
      A     "Zawsze_False";
      =     "Asi_output".Adres_8_bit_1;	//CC_Wise
//****************Wolno***********************
      A     "Zawsze_False";
      =     "Asi_output".Adres_8_bit_2;	//Wolno
//****************Bit_Bezpieczenstwa**********
      A     "Marka_Bezpieczenstwa";	//Safety
      =     "Asi_output".Adres_8_bit_3;
NETWORK
TITLE = Temporary placeholder variable
//Banda 9 Rolki
//****************ClockWise*******************
      A     "Zawsze_False";	//C_Wise
      =     "Asi_output".Adres_9_bit_0;
//****************CounterClockWise************
      A     "AIO".Banda_9.C_Wise;
      =     "Asi_output".Adres_9_bit_1;	//CC_Wise
//****************Wolno***********************
      A     "Zawsze_True";
      =     "Asi_output".Adres_9_bit_2;	//Wolno
//****************Bit_Bezpieczenstwa**********
      A     "Marka_Bezpieczenstwa";	//Safety
      =     "Asi_output".Adres_9_bit_3;
NETWORK
TITLE = Temporary placeholder variable
//Banda 10 Rolki
//Uwaga Banda ta nalezy do foliarki
//Sygnaly z foliarki
      A     "MPI_GD".IN.Motor_10_Lewo;
      =     "AIO".Banda_10.C_Wise;
      A     "MPI_GD".IN.Motor_10_Prawo;
      =     "AIO".Banda_10.CC_Wise;
//****************ClockWise*******************
      A     "AIO".Banda_10.C_Wise;	//C_Wise
      =     "Asi_output".Adres_10_bit_0;
//****************CounterClockWise************
      A     "AIO".Banda_10.CC_Wise;
      =     "Asi_output".Adres_10_bit_1;	//CC_Wise
//****************Wolno***********************
      A     "Zawsze_True";
      =     "Asi_output".Adres_10_bit_2;	//Wolno
//****************Bit_Bezpieczenstwa**********
      A     "Marka_Bezpieczenstwa";	//Safety
      =     "Asi_output".Adres_10_bit_3;
NETWORK
TITLE = Temporary placeholder variable
//Banda 11 Rolki
//Uwaga Banda ta nalezy do foliarki
//Sygnaly z foliarki
      A     "MPI_GD".IN.Motor_11_Lewo;
      =     "AIO".Banda_11.C_Wise;
      A     "MPI_GD".IN.Motor_11_Prawo;
      =     "AIO".Banda_11.CC_Wise;
//****************ClockWise*******************
      A     "AIO".Banda_11.C_Wise;	//C_Wise
      =     "Asi_output".Adres_11_bit_0;
//****************CounterClockWise************
      A     "AIO".Banda_11.CC_Wise;
      =     "Asi_output".Adres_11_bit_1;	//CC_Wise
//****************Wolno***********************
      A     "Zawsze_True";
      =     "Asi_output".Adres_11_bit_2;	//Wolno
//****************Bit_Bezpieczenstwa**********
      A     "Marka_Bezpieczenstwa";	//Safety
      =     "Asi_output".Adres_11_bit_3;
NETWORK
TITLE = Temporary placeholder variable
//Banda 12 Rolki wlot 2 na obrotnice
//****************ClockWise*******************
      A     "AIO".Banda_12.C_Wise;	//C_Wise
      =     "Asi_output".Adres_12_bit_0;
//****************CounterClockWise************
      A     "Zawsze_False";
      =     "Asi_output".Adres_12_bit_1;	//CC_Wise
//****************Wolno***********************
      A     "Zawsze_False";
      =     "Asi_output".Adres_12_bit_2;	//Wolno
//****************Bit_Bezpieczenstwa**********
      A     "Marka_Bezpieczenstwa";	//Safety
      =     "Asi_output".Adres_12_bit_3;
NETWORK
TITLE = Temporary placeholder variable
//Banda 13 Adres 13 Rolki na obrotnicy
//****************ClockWise*******************
      A     "AIO".Banda_13.C_Wise;	//C_Wise
      =     "Asi_output".Adres_13_bit_0;
//****************CounterClockWise************
      A     "AIO".Banda_13.CC_Wise;
      =     "Asi_output".Adres_13_bit_1;	//CC_Wise
//****************Wolno***********************
      A     "Zawsze_False";
      =     "Asi_output".Adres_13_bit_2;	//Wolno
//****************Bit_Bezpieczenstwa**********
      A     "Marka_Bezpieczenstwa";	//Safety
      =     "Asi_output".Adres_13_bit_3;
NETWORK
TITLE = Temporary placeholder variable
//Banda 14 Adres 14 Wylot z maszyny
//****************ClockWise*******************
      A     "AIO".Banda_14.C_Wise;	//C_Wise
      =     "Asi_output".Adres_14_bit_0;
//****************CounterClockWise************
      A     "Zawsze_False";
      =     "Asi_output".Adres_14_bit_1;	//CC_Wise
//****************Wolno***********************
      A     "Zawsze_False";
      =     "Asi_output".Adres_14_bit_2;	//Wolno
//****************Bit_Bezpieczenstwa**********
      A     "Marka_Bezpieczenstwa";	//Safety
      =     "Asi_output".Adres_14_bit_3;
NETWORK
TITLE = Temporary placeholder variable
//Obrotnica 15 Adres 15
//****************ClockWise*******************
      A     "AIO".Obr_15.C_Wise;
      =     "Asi_output".Adres_15_bit_0;
//****************CounterClockWise************
      A     "AIO".Obr_15.CC_Wise;
      =     "Asi_output".Adres_15_bit_1;	//CC_Wise
//****************Wolno***********************
      AN    "AIO".Obr_15.Wolno;
      =     "Asi_output".Adres_15_bit_2;	//Wolno
//****************Bit_Bezpieczenstwa**********
      A     "Marka_Bezpieczenstwa";	//Safety
      =     "Asi_output".Adres_15_bit_3;
NETWORK
TITLE =
//adres 16 rygiel brak output
NETWORK
TITLE = Temporary placeholder variable
//adres 17 reset kurtyn
//****************Reset wlot *****************
      A     "AIO".Reset_17.Reset_Wlot;
      =     "Asi_output".Adres_17_bit_0;	//reset wlot
//****************Reset wylot ****************
      A     "AIO".Reset_17.Reset_Wylot;
      =     "Asi_output".Adres_17_bit_1;	//reset wylot
NETWORK
TITLE = Temporary placeholder variable
//Obrotnica 18  Adres 18
//****************ClockWise*******************
      A     "AIO".Obr_18.C_Wise;
      =     "Asi_output".Adres_18_bit_0;
//****************CounterClockWise************
      A     "AIO".Obr_18.CC_Wise;
      =     "Asi_output".Adres_18_bit_1;	//CC_Wise
//****************Wolno***********************
      A     "AIO".Obr_18.Wolno;
      =     "Asi_output".Adres_18_bit_2;	//Wolno
//****************Bit_Bezpieczenstwa**********
      A     "Marka_Bezpieczenstwa";	//Safety
      =     "Asi_output".Adres_18_bit_3;
NETWORK
TITLE = Temporary placeholder variable
//Adres 19 brak sygnalow output
NETWORK
TITLE = Temporary placeholder variable
//Obrotnica 20 Adres 20
//****************ClockWise*******************
      A     "AIO".Obr_20.C_Wise;
      =     "Asi_output".Adres_20_bit_0;
//****************CounterClockWise************
      A     "AIO".Obr_20.CC_Wise;
      =     "Asi_output".Adres_20_bit_1;	//CC_Wise
//****************Wolno***********************
      A     "AIO".Obr_20.Wolno;
      =     "Asi_output".Adres_20_bit_2;	//Wolno
//****************Bit_Bezpieczenstwa**********
      A     "Marka_Bezpieczenstwa";	//Safety
      =     "Asi_output".Adres_20_bit_3;
NETWORK
TITLE = Temporary placeholder variable
//Adres 21, 22 Brak Output
NETWORK
TITLE = Temporary placeholder variable
//Banda 23
//
//****************ClockWise*******************
      A     "AIO".Banda_23.CC_Wise;	//C_Wise
      =     "Asi_output".Adres_23_bit_0;
//****************CounterClockWise************
      A     "AIO".Banda_23.C_Wise;
      =     "Asi_output".Adres_23_bit_1;	//CC_Wise
//****************Wolno***********************
      A     "AIO".Banda_23.Wolno;
      =     "Asi_output".Adres_23_bit_2;	//Wolno
//****************Bit_Bezpieczenstwa**********
      A     "Marka_Bezpieczenstwa";	//Safety
      =     "Asi_output".Adres_23_bit_3;
NETWORK
TITLE = Temporary placeholder variable
//Banda 24
//
//****************ClockWise*******************
      A     "AIO".Banda_24.CC_Wise;	//C_Wise
      =     "Asi_output".Adres_24_bit_0;
//****************CounterClockWise************
      A     "AIO".Banda_24.C_Wise;
      =     "Asi_output".Adres_24_bit_1;	//CC_Wise
//****************Wolno***********************
      A     "Zawsze_True";
      =     "Asi_output".Adres_24_bit_2;	//Wolno
//****************Bit_Bezpieczenstwa**********
      A     "Marka_Bezpieczenstwa";	//Safety
      =     "Asi_output".Adres_24_bit_3;
NETWORK
TITLE =
//25,26 to kurtyny bezpieczenstwa brak output
NETWORK
TITLE =
//Aedrs 27,28,29,30,31. Adresy ESTOP brak syganlow output
NETWORK
TITLE =
//Dziekuje za uwage
END_FUNCTION

FUNCTION "Rejestr_Tasm" : VOID	// FC 30
VERSION : 0.1
BEGIN
NETWORK
TITLE =
//marki uzywane od mb60. 
//Palety sa przekazywane za pomoca rejstru przesuwnego bitowego
//Poczatek monitorowania
      O     "AIO".Banda_4.Foto_1;
      O     "AIO".Banda_4.Foto_2;
      A     "AIO".Banda_4.Potw_Dost_Wlot_2;
      S     M 60.0;
//Przekazanie na pierwsza bande (banda 5)
      A     "AIO".Banda_5.Foto_1;
      A     "AIO".Banda_5.Paleta_Dost_do_Pop;
      A     M 60.0;
      JCN   et_1;
      S     M 60.1;
      R     M 60.0;
et_1: NOP   0;
      A     "AIO".Banda_6.Foto_1;
      A     "AIO".Banda_6.Paleta_Dost_do_Pop;
      A     M 60.1;
      JCN   et_2;
      S     M 60.2;
      R     M 60.1;
et_2: NOP   0;
      A     "AIO".Banda_7.Foto_1;
      A     "AIO".Banda_7.Paleta_Dost_do_Pop;
      A     M 60.2;
      JCN   et_3;
      S     M 60.3;
      R     M 60.2;
et_3: NOP   0;
      A     "AIO".Banda_8.Foto_1;
      A     "AIO".Banda_8.Paleta_Dost_do_Pop;
      A     M 60.3;
      JCN   et_4;
      S     M 60.4;
      R     M 60.3;
et_4: NOP   0;
      A     "AIO".Banda_9.Foto_1;
      A     "AIO".Banda_9.Paleta_Dost_do_Pop;
      A     M 60.4;
      JCN   et_5;
      S     M 60.5;
      R     M 60.4;
et_5: NOP   0;
//Banda 10 to foliarka
      A     "AIO".Banda_10.Foto_1;
      A     "AIO".Banda_10.Paleta_Dost_do_Pop;
      A     M 60.5;
      JCN   et_6;
      S     M 60.6;
      R     M 60.5;
et_6: NOP   0;
      A     M 60.6;
      A     "MPI_GD".IN.Foto_Banda_1;	// run in 
      S     M 62.0;
      A     M 62.0;
      A     "MPI_GD".IN.Foto_Owijarka;	//foto banda 4
      JCN   et_7;
      S     M 66.7;
      R     M 66.6;
      R     M 66.2;
et_7: NOP   0;
      A     M 66.7;
      =     "MPI_GD".OUT.Zmien_Program_Na_4;
      A     "MPI_GD".IN.Rezerwa_1;
      R     M 66.7;
//nie gotowe wiec wszystkie foliowane
      SET;
      R     "MPI_GD".OUT.Zmien_Program_Na_4;
      R     "MPI_GD".OUT.Zmien_Pragram_Na_3;
END_FUNCTION

FUNCTION "FC_Auto_Reczny" : VOID	// FC 40
//Funkcja przelaczajaca miedzy auto i recznym
VERSION : 0.1
VAR_INPUT
  Enable : BOOL ;	//Zezwolenie na dzia³anie
  Reczny : BOOL ;
  Auto : BOOL ;
  Strefa_Bezp : BOOL ;
  Test_Lampek : BOOL ;	//test lampek
  Stop : BOOL ;
  Reset_1 : BOOL ;
  Reset_2 : BOOL ;
  Reset_3 : BOOL ;
END_VAR
VAR_OUTPUT
  Lampka_Reczny : BOOL ;
  Lampka_Auto : BOOL ;
END_VAR
VAR_IN_OUT
  Auto_Reczny : BOOL ;	//Auto 1, Reczny 0
END_VAR
BEGIN
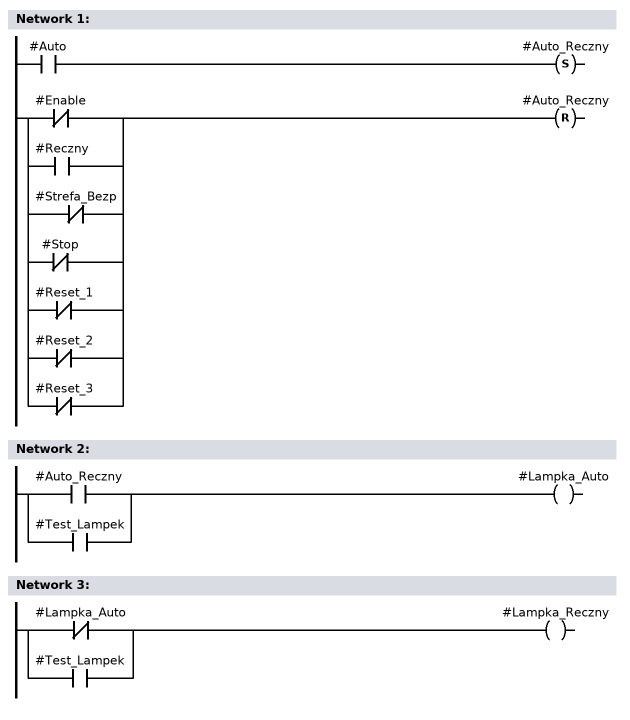
NETWORK
TITLE =
      A     #Auto;
      S     #Auto_Reczny;
      A(;
      ON    #Enable;
      O     #Reczny;
      ON    #Strefa_Bezp;
      ON    #Stop;
      ON    #Reset_1;
      ON    #Reset_2;
      ON    #Reset_3;
      );
      R     #Auto_Reczny;
      NOP   0;
NETWORK
TITLE =
      O     #Auto_Reczny;
      O     #Test_Lampek;
      =     #Lampka_Auto;
NETWORK
TITLE =
      ON    #Lampka_Auto;
      O     #Test_Lampek;
      =     #Lampka_Reczny;
END_FUNCTION

FUNCTION "Przycisk_Reset" : VOID	// FC 41
//Funkcja sluzy do jednoczesnej oblugi bledow oraz kasowania aktualnego kroku. 
//-Jezeli wcisnie sie przycisk to krotko do 5s to nastopi pruba kasowania bledu.
//-Jezeli wcisnie sie przycisk dlugo powyzej 5s to nastapi szybkie migniecie i 
//reset krokow
//
VERSION : 0.1
VAR_INPUT
  i_PB_Reset : BOOL ;
  i_T1 : TIMER ;	//Timer do dlugiego resetowania
  i_Czas_Trzymania : S5TIME ;
  i_T2 : TIMER ;	//Timer migania po przycisku
  i_Stop_Maszyny : BOOL ;
  i_Czas_Potw_Reset : S5TIME ;
  i_Clock : BOOL ;	//Zegar 100ms
END_VAR
VAR_OUTPUT
  o_Lampka_Reset : BOOL ;
END_VAR
VAR_IN_OUT
  o_Reset_Bledu : BOOL ;
  o_Reset_Krokow : BOOL ;
  io_Blok : BOOL ;
END_VAR
VAR_TEMP
  Temp_Help_1 : BOOL ;
  Temp_Help_2 : BOOL ;
END_VAR
BEGIN
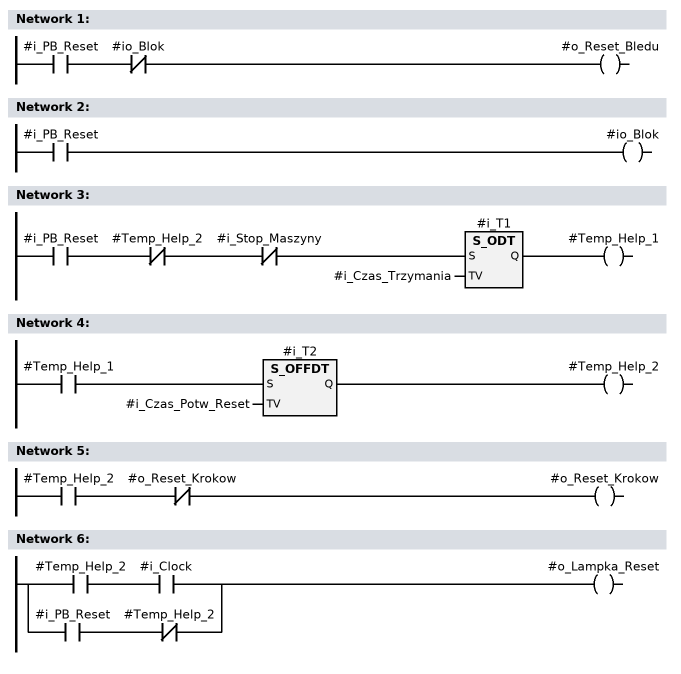
NETWORK
TITLE =
      A     #i_PB_Reset;
      AN    #io_Blok;
      =     #o_Reset_Bledu;
NETWORK
TITLE =
      A     #i_PB_Reset;
      =     #io_Blok;
NETWORK
TITLE =
      A     #i_PB_Reset;
      AN    #Temp_Help_2;
      AN    #i_Stop_Maszyny;
      L     #i_Czas_Trzymania;
      SD    #i_T1;
      NOP   0;
      NOP   0;
      NOP   0;
      A     #i_T1;
      =     #Temp_Help_1;
NETWORK
TITLE =
      A     #Temp_Help_1;
      L     #i_Czas_Potw_Reset;
      SF    #i_T2;
      NOP   0;
      NOP   0;
      NOP   0;
      A     #i_T2;
      =     #Temp_Help_2;
NETWORK
TITLE =
//Reset krokow
      A     #Temp_Help_2;
      AN    #o_Reset_Krokow;
      =     #o_Reset_Krokow;
NETWORK
TITLE =
//Lampka reset
      A     #Temp_Help_2;
      A     #i_Clock;
      O;
      A     #i_PB_Reset;
      AN    #Temp_Help_2;
      =     #o_Lampka_Reset;
END_FUNCTION

FUNCTION "Obrotnica_Na_Pozycje" : VOID	// FC 51
VERSION : 0.1
VAR_INPUT
  Jedz_Na_0st : BOOL ;
  Jedz_Na_90st : BOOL ;
  Czujnik_90st : BOOL ;
  Czujnik_0st : BOOL ;
  Czujnik_Ham_90st : BOOL ;
  Czujnik_Ham_0st : BOOL ;
  Odblowuj_Obrotnice : BOOL ;
END_VAR
VAR_OUTPUT
  Na_Pozycji_0st : BOOL ;	//Obrotnica na pozycji 0 stopni
  Na_Pozycji_90st : BOOL ;	//Obrotnica na pozycji 90 stopni
  Motor_Wolno : BOOL ;
  Odblokowanie_Rolek : BOOL ;
END_VAR
VAR_IN_OUT
  Talerz_w_Lewo : BOOL ;
  Talerz_w_Prawo : BOOL ;
END_VAR
BEGIN
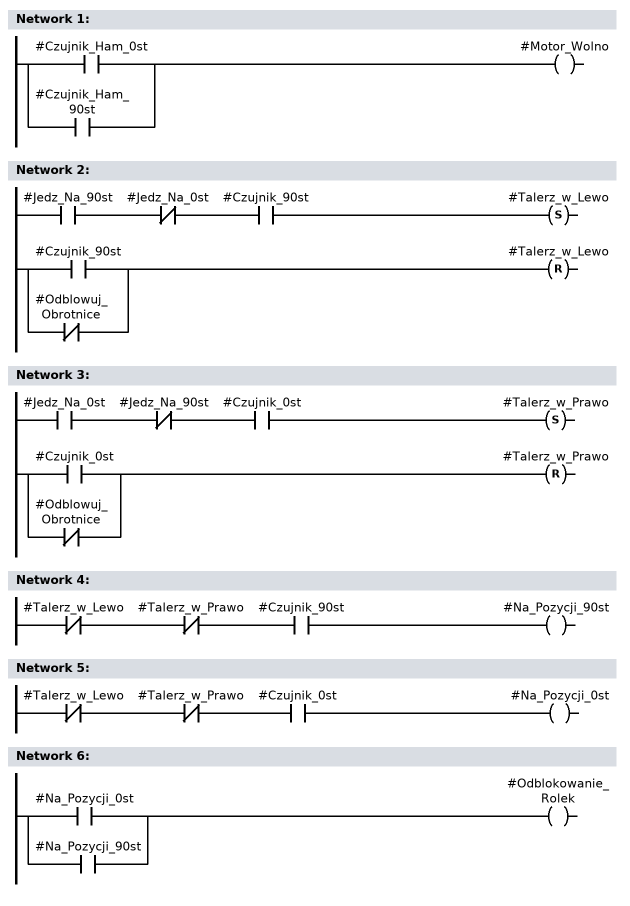
NETWORK
TITLE =
//Motor wolno gdy czujniki hamowania
      O     #Czujnik_Ham_0st;
      O     #Czujnik_Ham_90st;
      =     #Motor_Wolno;
NETWORK
TITLE =
      A     #Jedz_Na_90st;
      AN    #Jedz_Na_0st;
      A     #Czujnik_90st;
      S     #Talerz_w_Lewo;
      A(;
      O     #Czujnik_90st;
      ON    #Odblowuj_Obrotnice;
      );
      R     #Talerz_w_Lewo;
      NOP   0;
NETWORK
TITLE =
      A     #Jedz_Na_0st;
      AN    #Jedz_Na_90st;
      A     #Czujnik_0st;
      S     #Talerz_w_Prawo;
      A(;
      O     #Czujnik_0st;
      ON    #Odblowuj_Obrotnice;
      );
      R     #Talerz_w_Prawo;
      NOP   0;
NETWORK
TITLE =
      AN    #Talerz_w_Lewo;
      AN    #Talerz_w_Prawo;
      A     #Czujnik_90st;
      =     #Na_Pozycji_90st;
NETWORK
TITLE =
      AN    #Talerz_w_Lewo;
      AN    #Talerz_w_Prawo;
      A     #Czujnik_0st;
      =     #Na_Pozycji_0st;
NETWORK
TITLE =
//Odblokowanie napedu rolkowego
      O     #Na_Pozycji_0st;
      O     #Na_Pozycji_90st;
      =     #Odblokowanie_Rolek;
END_FUNCTION

FUNCTION "ASI_Odczyt" : VOID	// FC 80
//Pobieranie danych z modulu ASI CP 342-2
AUTHOR : Kng
FAMILY : Asi_fun
NAME : r_ASi
VERSION : 0.1
VAR_INPUT
  CP_Adr : INT ;
  DB_Nr : INT ;
END_VAR
VAR_TEMP
  L_CP_Adr : DWORD ;
  L_DB_Target : WORD ;
  L_Start_Adr : DWORD ;
  L_Count : WORD ;
  Word_CP_Adr : WORD ;
  Fault : INT ;
  Target : ANY ;
END_VAR
BEGIN
NETWORK
TITLE =
      L     #CP_Adr;	// Adres urzadzenia
      SLD   3;	//Przejscie na wskaznik
      T     #L_CP_Adr;
      L     #DB_Nr;	// Nr bloku db
      T     #L_DB_Target;
      L     0;	// Start adres db 
      SLD   3;	// Przejscie na wskaznik
      T     #L_Start_Adr;
      L     4;	// Liczba petli (pobranie 16 bajtow)
next: T     #L_Count;
      L     PID [#L_CP_Adr];	// Zaladowanie wejsc
      OPN   DB [#L_DB_Target];	// Otwarcie db
      T     DBD [#L_Start_Adr];	// Wgranie danych
      L     #L_CP_Adr;	// Zaladuj adres cp
      SRD   3;	// przejscie na format obliczen
      L     4;
      +I;	// bo doble word 
      SLD   3;	// Przejscie na wskaznik
      T     #L_CP_Adr;
      L     #L_Start_Adr;	// Przesuniecie bloku danych
      SRD   3;	// do nastepnego ladowania
      L     4;
      +I;	// 
      SLD   3;	// 
      T     #L_Start_Adr;
      L     #L_Count;
      LOOP  next;	// powrot petli  next
NETWORK
TITLE =
//Recnum nie wiem co to jest dana z kart katologowych
//Funkcja ta odpowiada za segment adresowania B
      LAR1  P##Target;	// wskaznik do obszaru  docelowego
      L     W#16#1002;	//zaladuj skladnie 10 i typ byte 02
      T     LW [AR1,P#0.0];
      L     16;	//zaladuj dl. obszaru do kopiowania
      T     LW [AR1,P#2.0];
      L     #DB_Nr;	//zaladuj nr bloku db (np.:db33)
      T     LW [AR1,P#4.0];
      L     16;	//zaladuj start_adres odbioru danych
      SLD   3;	// przesun w lewo (bit ostatni ma 0.0
      OD    DW#16#84000000;	//ustaw wartosc 84-db
      T     LD [AR1,P#6.0];
//------------------------------------
      L     #CP_Adr;
      T     #Word_CP_Adr;
      CALL  "RD_REC" (
           REQ                      := TRUE,
           IOID                     := B#16#54,
           LADDR                    := #Word_CP_Adr,
           RECNUM                   := B#16#96,
           RET_VAL                  := #Fault,
           BUSY                     := L 16.1,
           RECORD                   := #Target);
END_FUNCTION

FUNCTION "ASI_Zapis" : VOID	// FC 81
//Wgranie danych do modulu ASI CP 342-2
//Funkcja ta powinna znalezc sie po programie przypiania wyjsc!!!!
AUTHOR : Kng
FAMILY : Asi_fun
NAME : w_ASi
VERSION : 0.1
VAR_INPUT
  CP_Adr : INT ;	//Adres modulu cp343-2
  DB_Nr : INT ;	//Nr db z ktorego pobierane dane
END_VAR
VAR_TEMP
  L_CP_Adr : DWORD ;
  L_DB_Target : WORD ;
  L_Start_Adr : DWORD ;
  L_Count : WORD ;
  Word_CP_Adr : WORD ;
  Fault : INT ;
  Source : ANY ;
END_VAR
BEGIN
NETWORK
TITLE =
      L     #CP_Adr;	// Adres urzadzenia
      SLD   3;	//Przejscie na wskaznik
      T     #L_CP_Adr;
      L     #DB_Nr;	// Nr bloku db
      T     #L_DB_Target;
      L     0;	// Start adres db 
      SLD   3;	// Przejscie na wskaznik
      T     #L_Start_Adr;
      L     4;	// Liczba petli (pobranie 16 bajtow)
next: T     #L_Count;
      OPN   DB [#L_DB_Target];	// Otwarcie db
      L     DBD [#L_Start_Adr];	// Zaladowanie danych
      T     PQD [#L_CP_Adr];	// Wgranie wyjsc
      L     #L_CP_Adr;	// Zaladuj adres cp
      SRD   3;	// przejscie na format obliczen
      L     4;
      +I;	// bo double word 
      SLD   3;	// Przejscie na wskaznik
      T     #L_CP_Adr;
      L     #L_Start_Adr;	// Przesuniecie bloku danych
      SRD   3;	// do nastepnego ladowania
      L     4;
      +I;	// 
      SLD   3;	// 
      T     #L_Start_Adr;
      L     #L_Count;
      LOOP  next;	// powrot petli  next
//mala maszyna to dodac beu
NETWORK
TITLE =
//Recnum nie wiem co to jest dana z kart katologowych
//Funkcja ta odpowiada za segment adresowania B
      LAR1  P##Source;	// wskaznik do obszaru  pobierajacego
      L     W#16#1002;	//zaladuj skladnie 10 i typ byte 02
      T     LW [AR1,P#0.0];
      L     16;	//zaladuj dl. obszaru do kopiowania
      T     LW [AR1,P#2.0];
      L     #DB_Nr;	//zaladuj nr bloku db (np.:db33)
      T     LW [AR1,P#4.0];
      L     16;	//zaladuj start_adres odbioru danych
      SLD   3;	// przesun w lewo (bit ostatni ma 0.0
      OD    DW#16#84000000;	//ustaw wartosc 84-db
      T     LD [AR1,P#6.0];
//------------------------------------
      L     #CP_Adr;
      T     #Word_CP_Adr;
      CALL  "WR_REC" (
           REQ                      := TRUE,
           IOID                     := B#16#55,
           LADDR                    := #Word_CP_Adr,
           RECNUM                   := B#16#96,
           RECORD                   := #Source,
           RET_VAL                  := #Fault,
           BUSY                     := L 16.1);
END_FUNCTION

FUNCTION "Opoznienie_Wylotu" : VOID	// FC 85
VERSION : 0.1
VAR_INPUT
  Wejscie : BOOL ;	//Fotokomorka
  Timmer_1 : TIMER ;
  Timmer_2 : TIMER ;
END_VAR
VAR_OUTPUT
  Wyjscie : BOOL ;
END_VAR
VAR_IN_OUT
  Zmienna : BOOL ;
END_VAR
BEGIN
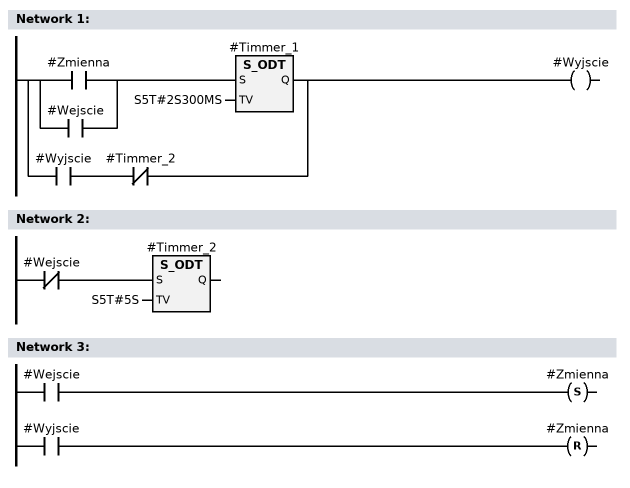
NETWORK
TITLE =
      O(;
      A(;
      O     #Zmienna;
      O     #Wejscie;
      );
      L     S5T#2S300MS;
      SD    #Timmer_1;
      NOP   0;
      NOP   0;
      NOP   0;
      A     #Timmer_1;
      );
      O;
      A     #Wyjscie;
      AN    #Timmer_2;
      =     #Wyjscie;
NETWORK
TITLE =
      AN    #Wejscie;
      L     S5T#5S;
      SD    #Timmer_2;
      NOP   0;
      NOP   0;
      NOP   0;
      NOP   0;
NETWORK
TITLE =
      A     #Wejscie;
      S     #Zmienna;
      A     #Wyjscie;
      R     #Zmienna;
      NOP   0;
END_FUNCTION

FUNCTION "Opoznienie_Wlotu" : VOID	// FC 86
VERSION : 0.1
VAR_INPUT
  Wejscie : BOOL ;	//Fotokomorka
  Timmer_1 : TIMER ;
  Timmer_2 : TIMER ;
END_VAR
VAR_OUTPUT
  Wyjscie : BOOL ;
END_VAR
VAR_IN_OUT
  Zmienna : BOOL ;
END_VAR
BEGIN
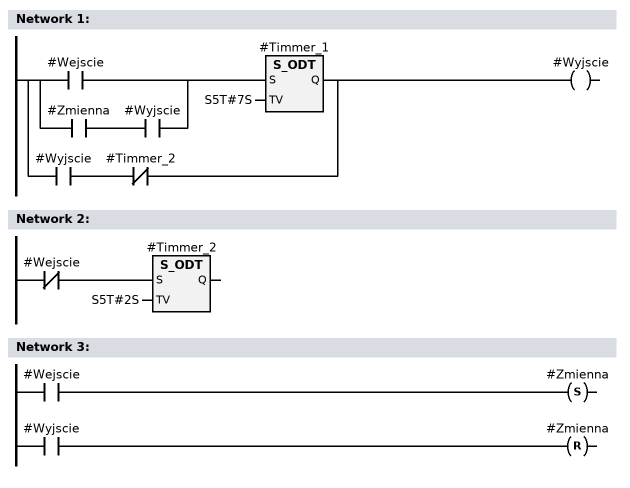
NETWORK
TITLE =
//Obecnosc palety jest aktywowana po 30s 
      O(;
      A(;
      O     #Wejscie;
      O;
      A     #Zmienna;
      A     #Wyjscie;
      );
      L     S5T#7S;
      SD    #Timmer_1;
      NOP   0;
      NOP   0;
      NOP   0;
      A     #Timmer_1;
      );
      O;
      A     #Wyjscie;
      AN    #Timmer_2;
      =     #Wyjscie;
NETWORK
TITLE =
//Filter 2s na fotokomorke aby nie zgasla gdy paleta jest na bandzie
      AN    #Wejscie;
      L     S5T#2S;
      SD    #Timmer_2;
      NOP   0;
      NOP   0;
      NOP   0;
      NOP   0;
NETWORK
TITLE =
      A     #Wejscie;
      S     #Zmienna;
      A     #Wyjscie;
      R     #Zmienna;
      NOP   0;
END_FUNCTION

FUNCTION "Opoznienie_Wlotu_2" : VOID	// FC 87
VERSION : 0.1
VAR_INPUT
  Wejscie : BOOL ;	//Fotokomorka
  Timmer_1 : TIMER ;
  Timmer_2 : TIMER ;
  Czas_Opoznienia : S5TIME ;
END_VAR
VAR_OUTPUT
  Wyjscie : BOOL ;
END_VAR
VAR_IN_OUT
  Zmienna : BOOL ;
END_VAR
BEGIN
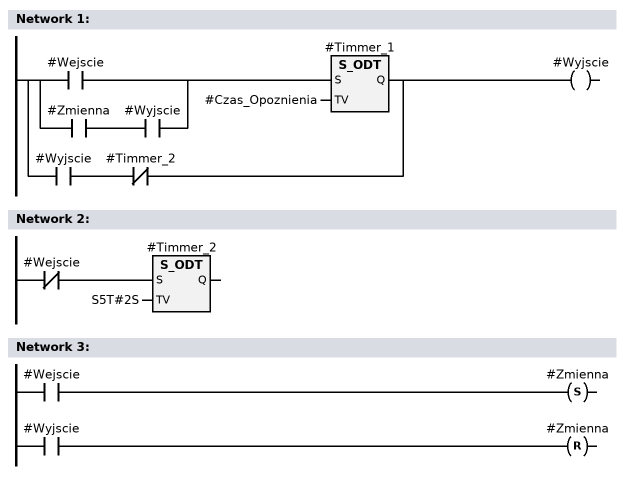
NETWORK
TITLE =
//Obecnosc palety jest aktywowana po 30s 
      O(;
      A(;
      O     #Wejscie;
      O;
      A     #Zmienna;
      A     #Wyjscie;
      );
      L     #Czas_Opoznienia;
      SD    #Timmer_1;
      NOP   0;
      NOP   0;
      NOP   0;
      A     #Timmer_1;
      );
      O;
      A     #Wyjscie;
      AN    #Timmer_2;
      =     #Wyjscie;
NETWORK
TITLE =
//Filter 2s na fotokomorke aby nie zgasla gdy paleta jest na bandzie
      AN    #Wejscie;
      L     S5T#2S;
      SD    #Timmer_2;
      NOP   0;
      NOP   0;
      NOP   0;
      NOP   0;
NETWORK
TITLE =
      A     #Wejscie;
      S     #Zmienna;
      A     #Wyjscie;
      R     #Zmienna;
      NOP   0;
END_FUNCTION

FUNCTION "Komunikacja_GD" : VOID	// FC 100
VERSION : 0.1
BEGIN
NETWORK
TITLE =
//Ten network celowo jest wolny
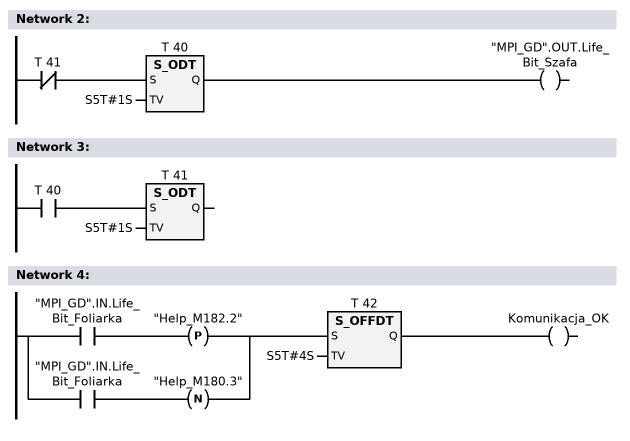
NETWORK
TITLE =
//Generator bit zycia foliarki
      AN    T 41;
      L     S5T#1S;
      SD    T 40;
      NOP   0;
      NOP   0;
      NOP   0;
      A     T 40;
      =     "MPI_GD".OUT.Life_Bit_Szafa;
NETWORK
TITLE =
//Generator bit zycia foliarki
      A     T 40;
      L     S5T#1S;
      SD    T 41;
      NOP   0;
      NOP   0;
      NOP   0;
      NOP   0;
NETWORK
TITLE =
//Sprawdzenie komunikacji z szafa transportera
      A(;
      A     "MPI_GD".IN.Life_Bit_Foliarka;
      FP    "Help_M182.2";
      O(;
      A     "MPI_GD".IN.Life_Bit_Foliarka;
      FN    "Help_M180.3";
      );
      );
      L     S5T#4S;
      SF    T 42;
      NOP   0;
      NOP   0;
      NOP   0;
      A     T 42;
      =     "Komunikacja_OK";
END_FUNCTION

FUNCTION "Obsluga bledow" : VOID	// FC 119
VERSION : 0.1
BEGIN
NETWORK
TITLE =
//Ten network celowo jest wolny
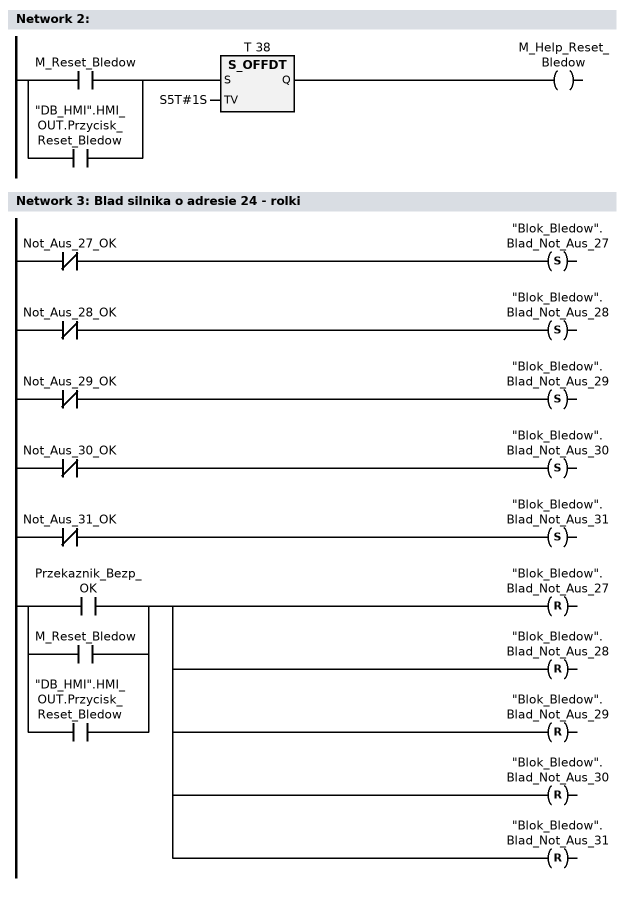
NETWORK
TITLE =
      A(;
      O     "M_Reset_Bledow";
      O     "DB_HMI".HMI_OUT.Przycisk_Reset_Bledow;
      );
      L     S5T#1S;
      SF    T 38;
      NOP   0;
      NOP   0;
      NOP   0;
      A     T 38;
      =     "M_Help_Reset_Bledow";
NETWORK
TITLE = Blad silnika o adresie 24 - rolki
//Bledy do panelu HMI
//Not Aus 27*******************************
      AN    "Not_Aus_27_OK";
      S     "Blok_Bledow".Blad_Not_Aus_27;
//Not Aus 28*******************************
      AN    "Not_Aus_28_OK";
      S     "Blok_Bledow".Blad_Not_Aus_28;
//Not Aus 29*******************************
      AN    "Not_Aus_29_OK";
      S     "Blok_Bledow".Blad_Not_Aus_29;
//Not Aus 30*******************************
      AN    "Not_Aus_30_OK";
      S     "Blok_Bledow".Blad_Not_Aus_30;
//Not Aus 31*******************************
      AN    "Not_Aus_31_OK";
      S     "Blok_Bledow".Blad_Not_Aus_31;
//Reset bledow not-aus
      O     "Przekaznik_Bezp_OK";
      O     "M_Reset_Bledow";
      O     "DB_HMI".HMI_OUT.Przycisk_Reset_Bledow;
      R     "Blok_Bledow".Blad_Not_Aus_27;
      R     "Blok_Bledow".Blad_Not_Aus_28;
      R     "Blok_Bledow".Blad_Not_Aus_29;
      R     "Blok_Bledow".Blad_Not_Aus_30;
      R     "Blok_Bledow".Blad_Not_Aus_31;
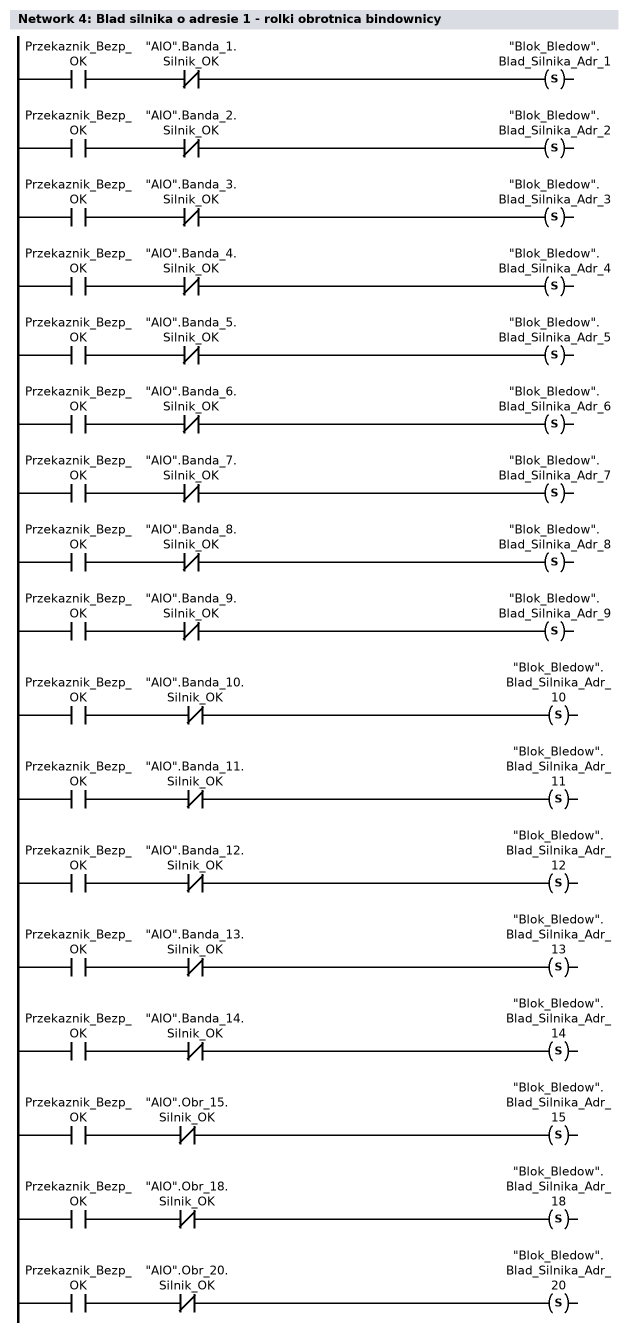
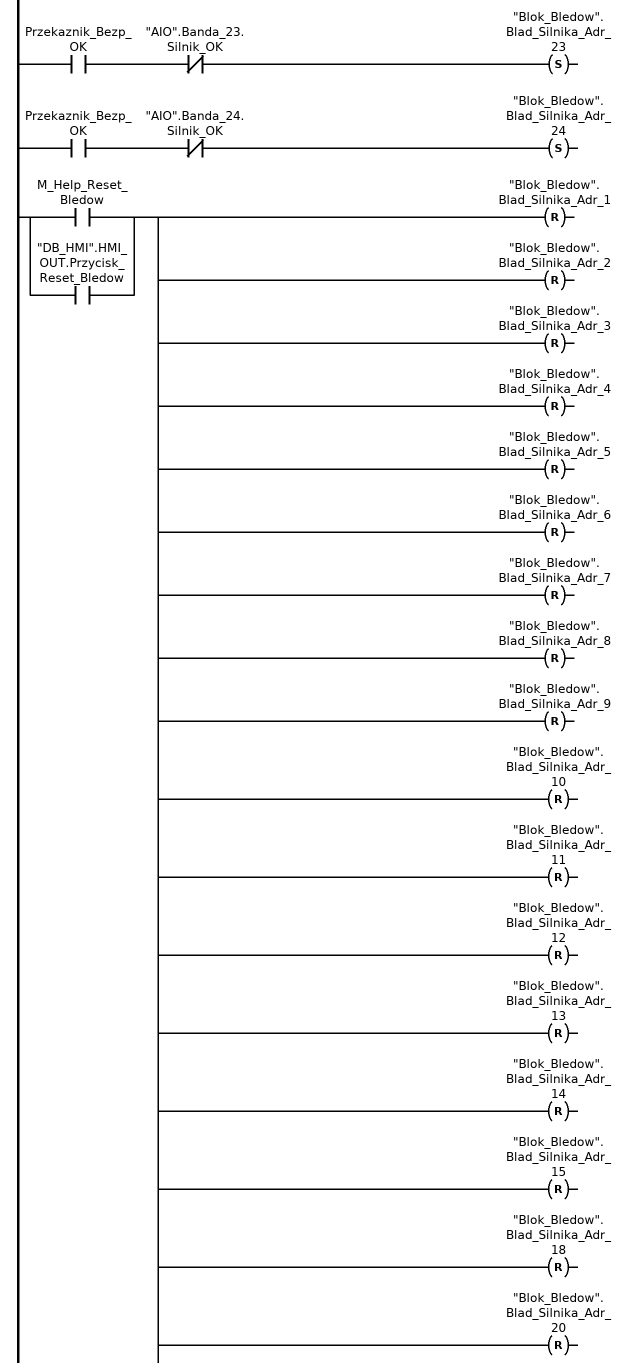
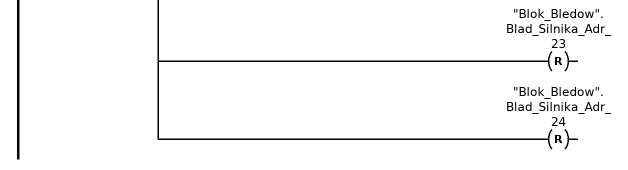
NETWORK
TITLE = Blad silnika o adresie 1 - rolki obrotnica bindownicy
//Bledy napedow
//Bledy napedow
      A     "Przekaznik_Bezp_OK";
      AN    "AIO".Banda_1.Silnik_OK;
      S     "Blok_Bledow".Blad_Silnika_Adr_1;
      A     "Przekaznik_Bezp_OK";
      AN    "AIO".Banda_2.Silnik_OK;
      S     "Blok_Bledow".Blad_Silnika_Adr_2;
      A     "Przekaznik_Bezp_OK";
      AN    "AIO".Banda_3.Silnik_OK;
      S     "Blok_Bledow".Blad_Silnika_Adr_3;
      A     "Przekaznik_Bezp_OK";
      AN    "AIO".Banda_4.Silnik_OK;
      S     "Blok_Bledow".Blad_Silnika_Adr_4;
      A     "Przekaznik_Bezp_OK";
      AN    "AIO".Banda_5.Silnik_OK;
      S     "Blok_Bledow".Blad_Silnika_Adr_5;
      A     "Przekaznik_Bezp_OK";
      AN    "AIO".Banda_6.Silnik_OK;
      S     "Blok_Bledow".Blad_Silnika_Adr_6;
      A     "Przekaznik_Bezp_OK";
      AN    "AIO".Banda_7.Silnik_OK;
      S     "Blok_Bledow".Blad_Silnika_Adr_7;
      A     "Przekaznik_Bezp_OK";
      AN    "AIO".Banda_8.Silnik_OK;
      S     "Blok_Bledow".Blad_Silnika_Adr_8;
      A     "Przekaznik_Bezp_OK";
      AN    "AIO".Banda_9.Silnik_OK;
      S     "Blok_Bledow".Blad_Silnika_Adr_9;
      A     "Przekaznik_Bezp_OK";
      AN    "AIO".Banda_10.Silnik_OK;
      S     "Blok_Bledow".Blad_Silnika_Adr_10;
      A     "Przekaznik_Bezp_OK";
      AN    "AIO".Banda_11.Silnik_OK;
      S     "Blok_Bledow".Blad_Silnika_Adr_11;
      A     "Przekaznik_Bezp_OK";
      AN    "AIO".Banda_12.Silnik_OK;
      S     "Blok_Bledow".Blad_Silnika_Adr_12;
      A     "Przekaznik_Bezp_OK";
      AN    "AIO".Banda_13.Silnik_OK;
      S     "Blok_Bledow".Blad_Silnika_Adr_13;
      A     "Przekaznik_Bezp_OK";
      AN    "AIO".Banda_14.Silnik_OK;
      S     "Blok_Bledow".Blad_Silnika_Adr_14;
      A     "Przekaznik_Bezp_OK";
      AN    "AIO".Obr_15.Silnik_OK;
      S     "Blok_Bledow".Blad_Silnika_Adr_15;
      A     "Przekaznik_Bezp_OK";
      AN    "AIO".Obr_18.Silnik_OK;
      S     "Blok_Bledow".Blad_Silnika_Adr_18;
      A     "Przekaznik_Bezp_OK";
      AN    "AIO".Obr_20.Silnik_OK;
      S     "Blok_Bledow".Blad_Silnika_Adr_20;
      A     "Przekaznik_Bezp_OK";
      AN    "AIO".Banda_23.Silnik_OK;
      S     "Blok_Bledow".Blad_Silnika_Adr_23;
      A     "Przekaznik_Bezp_OK";
      AN    "AIO".Banda_24.Silnik_OK;
      S     "Blok_Bledow".Blad_Silnika_Adr_24;
//Reset bledow napedow
//Reset bledow not-aus
      O     "M_Help_Reset_Bledow";
      O     "DB_HMI".HMI_OUT.Przycisk_Reset_Bledow;
      R     "Blok_Bledow".Blad_Silnika_Adr_1;
      R     "Blok_Bledow".Blad_Silnika_Adr_2;
      R     "Blok_Bledow".Blad_Silnika_Adr_3;
      R     "Blok_Bledow".Blad_Silnika_Adr_4;
      R     "Blok_Bledow".Blad_Silnika_Adr_5;
      R     "Blok_Bledow".Blad_Silnika_Adr_6;
      R     "Blok_Bledow".Blad_Silnika_Adr_7;
      R     "Blok_Bledow".Blad_Silnika_Adr_8;
      R     "Blok_Bledow".Blad_Silnika_Adr_9;
      R     "Blok_Bledow".Blad_Silnika_Adr_10;
      R     "Blok_Bledow".Blad_Silnika_Adr_11;
      R     "Blok_Bledow".Blad_Silnika_Adr_12;
      R     "Blok_Bledow".Blad_Silnika_Adr_13;
      R     "Blok_Bledow".Blad_Silnika_Adr_14;
      R     "Blok_Bledow".Blad_Silnika_Adr_15;
      R     "Blok_Bledow".Blad_Silnika_Adr_18;
      R     "Blok_Bledow".Blad_Silnika_Adr_20;
      R     "Blok_Bledow".Blad_Silnika_Adr_23;
      R     "Blok_Bledow".Blad_Silnika_Adr_24;
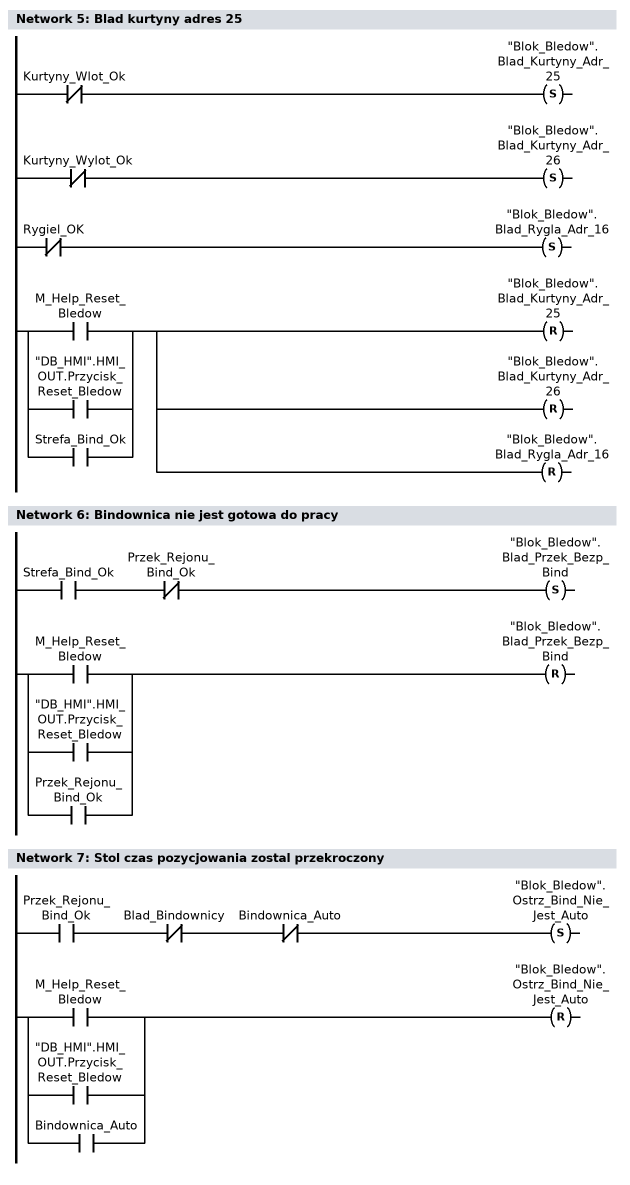
NETWORK
TITLE = Blad kurtyny adres 25
//Bledy kurtyn kasownie samoistne
      AN    "Kurtyny_Wlot_Ok";
      S     "Blok_Bledow".Blad_Kurtyny_Adr_25;
      AN    "Kurtyny_Wylot_Ok";
      S     "Blok_Bledow".Blad_Kurtyny_Adr_26;
      AN    "Rygiel_OK";
      S     "Blok_Bledow".Blad_Rygla_Adr_16;
      O     "M_Help_Reset_Bledow";
      O     "DB_HMI".HMI_OUT.Przycisk_Reset_Bledow;
      O     "Strefa_Bind_Ok";
      R     "Blok_Bledow".Blad_Kurtyny_Adr_25;
      R     "Blok_Bledow".Blad_Kurtyny_Adr_26;
      R     "Blok_Bledow".Blad_Rygla_Adr_16;
NETWORK
TITLE = Bindownica nie jest gotowa do pracy
//Blad Przekaznika bezpieczenstwa kurtyn
      A     "Strefa_Bind_Ok";
      AN    "Przek_Rejonu_Bind_Ok";
      S     "Blok_Bledow".Blad_Przek_Bezp_Bind;
      O     "M_Help_Reset_Bledow";
      O     "DB_HMI".HMI_OUT.Przycisk_Reset_Bledow;
      O     "Przek_Rejonu_Bind_Ok";
      R     "Blok_Bledow".Blad_Przek_Bezp_Bind;
NETWORK
TITLE = Stol czas pozycjowania zostal przekroczony
//Blad informacyjny bindownica nie jest w auto
      A     "Przek_Rejonu_Bind_Ok";
      AN    "Blad_Bindownicy";
      AN    "Bindownica_Auto";
      S     "Blok_Bledow".Ostrz_Bind_Nie_Jest_Auto;
      O     "M_Help_Reset_Bledow";
      O     "DB_HMI".HMI_OUT.Przycisk_Reset_Bledow;
      O     "Bindownica_Auto";
      R     "Blok_Bledow".Ostrz_Bind_Nie_Jest_Auto;
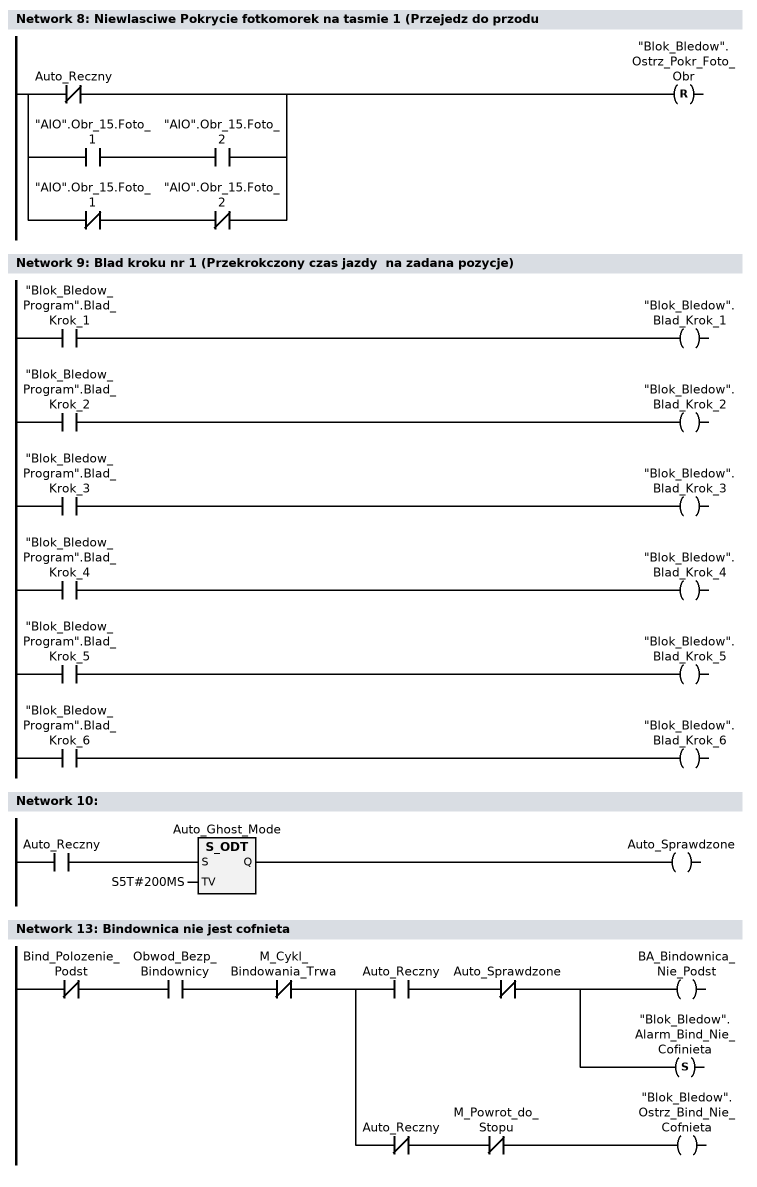
NETWORK
TITLE = Niewlasciwe Pokrycie fotkomorek na tasmie 1 (Przejedz do przodu 
//Ostrzezenie palety nie sa na fotokomorkach przednich
//
//Obrotnica
      ON    "Auto_Reczny";
      O;
      A     "AIO".Obr_15.Foto_1;
      A     "AIO".Obr_15.Foto_2;
      O;
      AN    "AIO".Obr_15.Foto_1;
      AN    "AIO".Obr_15.Foto_2;
      R     "Blok_Bledow".Ostrz_Pokr_Foto_Obr;
NETWORK
TITLE = Blad kroku nr 1 (Przekrokczony czas jazdy  na zadana pozycje)
//Bledy Zapalajaca czerwona lampke na panelu HMI
//Kwitowanie tych bledow przy pomocy przycisku. Reset nastepnie dalszy krok to 
//przywrocenie automatyki auto lub cyklem start
//
//
// Bledy czasu tranzycji krokow
      A     "Blok_Bledow_Program".Blad_Krok_1;
      =     "Blok_Bledow".Blad_Krok_1;
      A     "Blok_Bledow_Program".Blad_Krok_2;
      =     "Blok_Bledow".Blad_Krok_2;
      A     "Blok_Bledow_Program".Blad_Krok_3;
      =     "Blok_Bledow".Blad_Krok_3;
      A     "Blok_Bledow_Program".Blad_Krok_4;
      =     "Blok_Bledow".Blad_Krok_4;
      A     "Blok_Bledow_Program".Blad_Krok_5;
      =     "Blok_Bledow".Blad_Krok_5;
      A     "Blok_Bledow_Program".Blad_Krok_6;
      =     "Blok_Bledow".Blad_Krok_6;
NETWORK
TITLE =
//Wypadniecie maszyny z automatyki. Oraz powrot do polautomatu gdy automatyka nie 
//spelniona. 
      A     "Auto_Reczny";
      L     S5T#200MS;
      SD    "Auto_Ghost_Mode";
      NOP   0;
      NOP   0;
      NOP   0;
      A     "Auto_Ghost_Mode";
      =     "Auto_Sprawdzone";
NETWORK
TITLE =
NETWORK
TITLE =
//Warunki sprawdzane podczas 200ms trybu Ghost Mode
//bity m210 w gore
NETWORK
TITLE = Bindownica nie jest cofnieta
//Bindownica nie jest w pozycji podstawoej
      AN    "Bind_Polozenie_Podst";
      A     "Obwod_Bezp_Bindownicy";
      AN    "M_Cykl_Bindowania_Trwa";
      =     L 0.0;
      A     L 0.0;
      A     "Auto_Reczny";
      AN    "Auto_Sprawdzone";
      =     "BA_Bindownica_Nie_Podst";
      S     "Blok_Bledow".Alarm_Bind_Nie_Cofinieta;
      A     L 0.0;
      AN    "Auto_Reczny";
      AN    "M_Powrot_do_Stopu";
      =     "Blok_Bledow".Ostrz_Bind_Nie_Cofnieta;
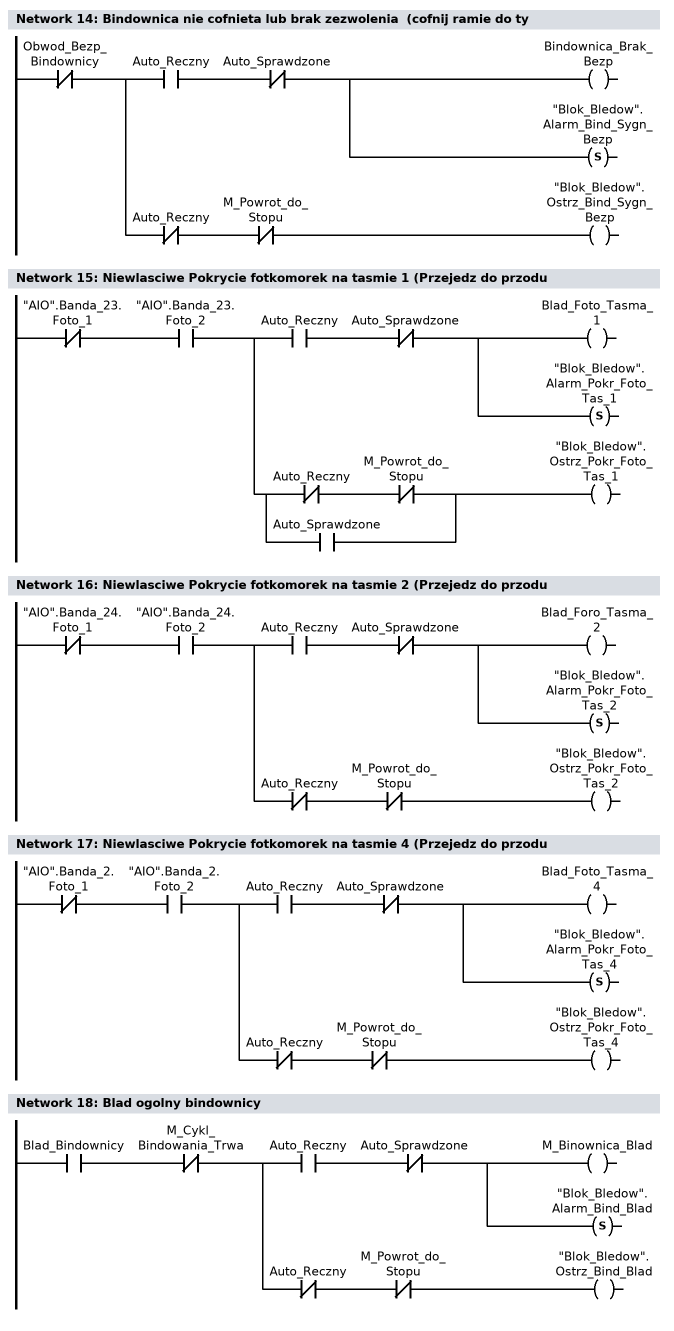
NETWORK
TITLE = Bindownica nie cofnieta lub brak zezwolenia  (cofnij ramie do ty
//Bindownica nie daje sygnalu bezpieczestwa
      AN    "Obwod_Bezp_Bindownicy";
      =     L 0.0;
      A     L 0.0;
      A     "Auto_Reczny";
      AN    "Auto_Sprawdzone";
      =     "Bindownica_Brak_Bezp";
      S     "Blok_Bledow".Alarm_Bind_Sygn_Bezp;
      A     L 0.0;
      AN    "Auto_Reczny";
      AN    "M_Powrot_do_Stopu";
      =     "Blok_Bledow".Ostrz_Bind_Sygn_Bezp;
NETWORK
TITLE = Niewlasciwe Pokrycie fotkomorek na tasmie 1 (Przejedz do przodu 
//Tasma 1 Wyjatek bo tutaj kladzie sie palete w automacie przez wozek
      AN    "AIO".Banda_23.Foto_1;
      A     "AIO".Banda_23.Foto_2;
      =     L 0.0;
      A     L 0.0;
      A     "Auto_Reczny";
      AN    "Auto_Sprawdzone";
      =     "Blad_Foto_Tasma_1";
      S     "Blok_Bledow".Alarm_Pokr_Foto_Tas_1;
      A     L 0.0;
      A(;
      AN    "Auto_Reczny";
      AN    "M_Powrot_do_Stopu";
      O     "Auto_Sprawdzone";
      );
      =     "Blok_Bledow".Ostrz_Pokr_Foto_Tas_1;
NETWORK
TITLE = Niewlasciwe Pokrycie fotkomorek na tasmie 2 (Przejedz do przodu 
//Tasma 2   O     "DB_HMI".HMI_OUT.Przycisk_Reset_Bledow
      AN    "AIO".Banda_24.Foto_1;
      A     "AIO".Banda_24.Foto_2;
      =     L 0.0;
      A     L 0.0;
      A     "Auto_Reczny";
      AN    "Auto_Sprawdzone";
      =     "Blad_Foro_Tasma_2";
      S     "Blok_Bledow".Alarm_Pokr_Foto_Tas_2;
      A     L 0.0;
      AN    "Auto_Reczny";
      AN    "M_Powrot_do_Stopu";
      =     "Blok_Bledow".Ostrz_Pokr_Foto_Tas_2;
NETWORK
TITLE = Niewlasciwe Pokrycie fotkomorek na tasmie 4 (Przejedz do przodu 
//Tasma:4      "DB_HMI".HMI_OUT.Przycisk_Reset_Bledow
      AN    "AIO".Banda_2.Foto_1;
      A     "AIO".Banda_2.Foto_2;
      =     L 0.0;
      A     L 0.0;
      A     "Auto_Reczny";
      AN    "Auto_Sprawdzone";
      =     "Blad_Foto_Tasma_4";
      S     "Blok_Bledow".Alarm_Pokr_Foto_Tas_4;
      A     L 0.0;
      AN    "Auto_Reczny";
      AN    "M_Powrot_do_Stopu";
      =     "Blok_Bledow".Ostrz_Pokr_Foto_Tas_4;
NETWORK
TITLE = Blad ogolny bindownicy 
//Blad ogolny bindownicy
      A     "Blad_Bindownicy";
      AN    "M_Cykl_Bindowania_Trwa";
      =     L 0.0;
      A     L 0.0;
      A     "Auto_Reczny";
      AN    "Auto_Sprawdzone";
      =     "M_Binownica_Blad";
      S     "Blok_Bledow".Alarm_Bind_Blad;
      A     L 0.0;
      AN    "Auto_Reczny";
      AN    "M_Powrot_do_Stopu";
      =     "Blok_Bledow".Ostrz_Bind_Blad;
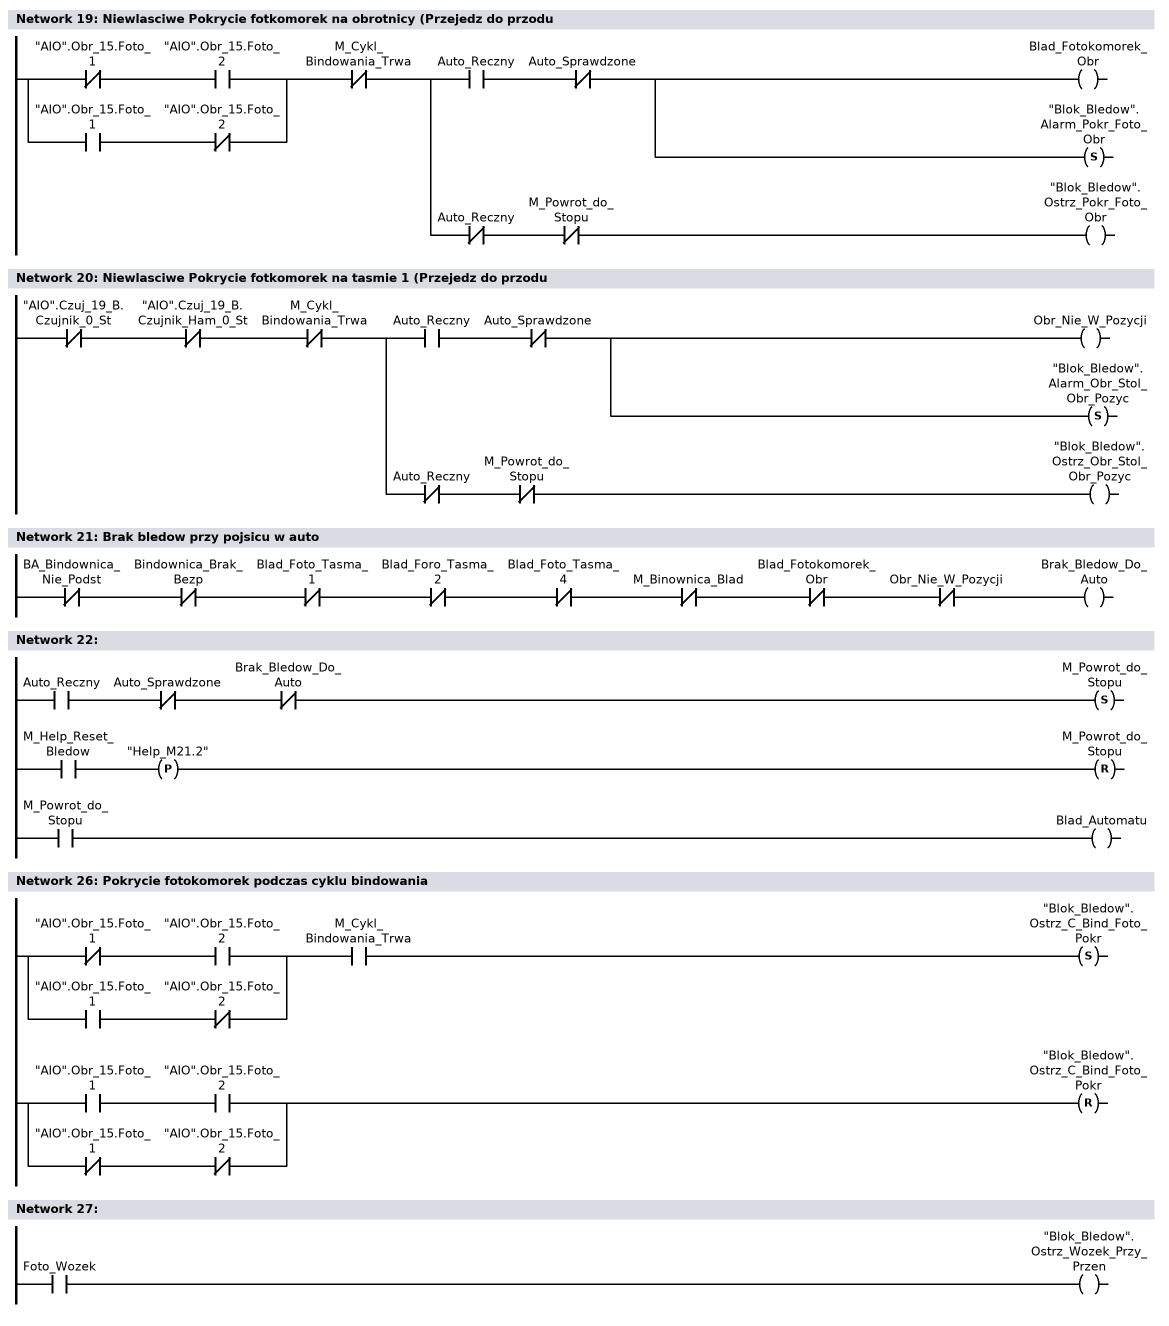
NETWORK
TITLE = Niewlasciwe Pokrycie fotkomorek na obrotnicy (Przejedz do przodu
//Blad fotokomorek stolu obrotowego
      A(;
      AN    "AIO".Obr_15.Foto_1;
      A     "AIO".Obr_15.Foto_2;
      O;
      A     "AIO".Obr_15.Foto_1;
      AN    "AIO".Obr_15.Foto_2;
      );
      AN    "M_Cykl_Bindowania_Trwa";
      =     L 0.0;
      A     L 0.0;
      A     "Auto_Reczny";
      AN    "Auto_Sprawdzone";
      =     "Blad_Fotokomorek_Obr";
      S     "Blok_Bledow".Alarm_Pokr_Foto_Obr;
      A     L 0.0;
      AN    "Auto_Reczny";
      AN    "M_Powrot_do_Stopu";
      =     "Blok_Bledow".Ostrz_Pokr_Foto_Obr;
NETWORK
TITLE = Niewlasciwe Pokrycie fotkomorek na tasmie 1 (Przejedz do przodu 
//Stol obrotowy nie w pozycji
      AN    "AIO".Czuj_19_B.Czujnik_0_St;
      AN    "AIO".Czuj_19_B.Czujnik_Ham_0_St;
      AN    "M_Cykl_Bindowania_Trwa";
      =     L 0.0;
      A     L 0.0;
      A     "Auto_Reczny";
      AN    "Auto_Sprawdzone";
      =     "Obr_Nie_W_Pozycji";
      S     "Blok_Bledow".Alarm_Obr_Stol_Obr_Pozyc;
      A     L 0.0;
      AN    "Auto_Reczny";
      AN    "M_Powrot_do_Stopu";
      =     "Blok_Bledow".Ostrz_Obr_Stol_Obr_Pozyc;
NETWORK
TITLE = Brak bledow przy pojsicu w auto
//Sprawdzam
      AN    "BA_Bindownica_Nie_Podst";
      AN    "Bindownica_Brak_Bezp";
      AN    "Blad_Foto_Tasma_1";
      AN    "Blad_Foro_Tasma_2";
      AN    "Blad_Foto_Tasma_4";
      AN    "M_Binownica_Blad";
      AN    "Blad_Fotokomorek_Obr";
      AN    "Obr_Nie_W_Pozycji";
      =     "Brak_Bledow_Do_Auto";
NETWORK
TITLE =
//Powrot do stopu polautomatu jesli jest blad
      A     "Auto_Reczny";
      AN    "Auto_Sprawdzone";
      AN    "Brak_Bledow_Do_Auto";
      S     "M_Powrot_do_Stopu";
      A     "M_Help_Reset_Bledow";
      FP    "Help_M21.2";
      R     "M_Powrot_do_Stopu";
      A     "M_Powrot_do_Stopu";
      =     "Blad_Automatu";
NETWORK
TITLE = Bindownica nie cofnieta lub brak zezwolenia  (cofnij ramie do ty
//reset komunikatow
//
      A     "M_Help_Reset_Bledow";
//Alarmy
      R     "Blok_Bledow".Alarm_Obr_Stol_Obr_Pozyc;
      R     "Blok_Bledow".Alarm_Bind_Nie_Cofinieta;
      R     "Blok_Bledow".Alarm_Bind_Sygn_Bezp;
      R     "Blok_Bledow".rez3;
      R     "Blok_Bledow".rez_6_0;
      R     "Blok_Bledow".Alarm_Pokr_Foto_Tas_1;
      R     "Blok_Bledow".Alarm_Pokr_Foto_Tas_2;
      R     "Blok_Bledow".Alarm_Pokr_Foto_Tas_4;
      R     "Blok_Bledow".Alarm_Pokr_Foto_Obr;
      R     "Blok_Bledow".Alarm_Bind_Nie_Jest_Auto;
      R     "Blok_Bledow".Alarm_Bind_Blad;
      R     "Blok_Bledow".rez_6_7;
      R     "Blok_Bledow".Ostrz_Prasa_Nie_W_Gorze;
      R     "Blok_Bledow".rez_7_1;
//Warnings
      R     "Blok_Bledow".Ostrz_Bind_Blad;
      R     "Blok_Bledow".Ostrz_Bind_Nie_Cofnieta;
      R     "Blok_Bledow".Ostrz_Bind_Sygn_Bezp;
      R     "Blok_Bledow".Ostrz_Bind_Nie_Jest_Auto;
      R     "Blok_Bledow".Ostrz_Stol_Obr_Foto;
      R     "Blok_Bledow".Ostrz_Obr_Stol_Obr_Pozyc;
      R     "Blok_Bledow".Ostrz_Pokr_Foto_Tas_1;
      R     "Blok_Bledow".Ostrz_Pokr_Foto_Tas_2;
      R     "Blok_Bledow".Ostrz_Pokr_Foto_Obr;
      R     "Blok_Bledow".Ostrz_Pokr_Foto_Tas_4;
      CLR;
NETWORK
TITLE =
//Koniec sprawdzanie wejscia w automatyke
NETWORK
TITLE =
//Sprawdzenie maszyny podczas cyklu. Zwracane sa ostrzezenia by byla informacja 
//ale nie przerwac dzialania
NETWORK
TITLE = Pokrycie fotokomorek podczas cyklu bindowania
//Niewlasciwe pokrycie fotokomorek podczas cyklu
      A(;
      AN    "AIO".Obr_15.Foto_1;
      A     "AIO".Obr_15.Foto_2;
      O;
      A     "AIO".Obr_15.Foto_1;
      AN    "AIO".Obr_15.Foto_2;
      );
      A     "M_Cykl_Bindowania_Trwa";
      S     "Blok_Bledow".Ostrz_C_Bind_Foto_Pokr;
      A(;
      A     "AIO".Obr_15.Foto_1;
      A     "AIO".Obr_15.Foto_2;
      O;
      AN    "AIO".Obr_15.Foto_1;
      AN    "AIO".Obr_15.Foto_2;
      );
      R     "Blok_Bledow".Ostrz_C_Bind_Foto_Pokr;
      NOP   0;
NETWORK
TITLE =
//Cykl trwa a bindownica nie jest z tylu
      A     "Foto_Wozek";
      =     "Blok_Bledow".Ostrz_Wozek_Przy_Przen;
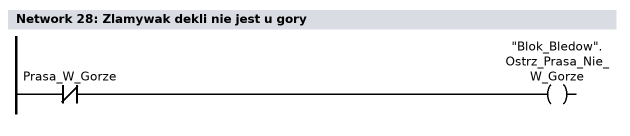
NETWORK
TITLE = Zlamywak dekli nie jest u gory 
      AN    "Prasa_W_Gorze";
      =     "Blok_Bledow".Ostrz_Prasa_Nie_W_Gorze;
END_FUNCTION

FUNCTION "FC_HMI" : VOID	// FC 120
VERSION : 0.1
VAR_TEMP
  LW0_Help : INT ;
END_VAR
BEGIN
NETWORK
TITLE =
//Ten network celowo wolny
NETWORK
TITLE = Tryb Pracy Wiazanie poprzeczne
//Wybranie trybu pracy resetuje pozostale tryby pracy
//1-Przelot
      A     "DB_HMI".HMI_IN_OUT.Tp_Przelot;
      R     "DB_HMI".HMI_IN_OUT.Tp_Wiazanie_Poprzeczne;
      R     "DB_HMI".HMI_IN_OUT.Tp_Wiazanie_Wzdluzne;
      R     "DB_HMI".HMI_IN_OUT.Tp_Wiazanie_Pop_Wzdl;
      R     "Blok_Para".Wiazanie_Poprzeczne;
      R     "Blok_Para".Wiazanie_Wzdluzne;
NETWORK
TITLE = Tryb Pracy Wiazanie poprzeczne
//Wybranie trybu pracy resetuje pozostale tryby pracy
//2-Wiazanie Poprzeczne
      A     "DB_HMI".HMI_IN_OUT.Tp_Wiazanie_Poprzeczne;
      R     "DB_HMI".HMI_IN_OUT.Tp_Przelot;
      R     "DB_HMI".HMI_IN_OUT.Tp_Wiazanie_Wzdluzne;
      R     "DB_HMI".HMI_IN_OUT.Tp_Wiazanie_Pop_Wzdl;
      S     "Blok_Para".Wiazanie_Poprzeczne;
      R     "Blok_Para".Wiazanie_Wzdluzne;
NETWORK
TITLE = Tryb Pracy Wiazanie poprzeczne
//Wybranie trybu pracy resetuje pozostale tryby pracy
//3-Wiazanie Wzdluzne
      A     "DB_HMI".HMI_IN_OUT.Tp_Wiazanie_Wzdluzne;
      R     "DB_HMI".HMI_IN_OUT.Tp_Przelot;
      R     "DB_HMI".HMI_IN_OUT.Tp_Wiazanie_Poprzeczne;
      R     "DB_HMI".HMI_IN_OUT.Tp_Wiazanie_Pop_Wzdl;
      R     "Blok_Para".Wiazanie_Poprzeczne;
      S     "Blok_Para".Wiazanie_Wzdluzne;
NETWORK
TITLE = Tryb Pracy Wiazanie poprzeczne
//Wybranie trybu pracy resetuje pozostale tryby pracy
//4-Wiazanie Poprzeczne i wzdluzne
      A     "DB_HMI".HMI_IN_OUT.Tp_Wiazanie_Pop_Wzdl;
      R     "DB_HMI".HMI_IN_OUT.Tp_Przelot;
      R     "DB_HMI".HMI_IN_OUT.Tp_Wiazanie_Poprzeczne;
      R     "DB_HMI".HMI_IN_OUT.Tp_Wiazanie_Wzdluzne;
      S     "Blok_Para".Wiazanie_Poprzeczne;
      S     "Blok_Para".Wiazanie_Wzdluzne;
NETWORK
TITLE = wybrano tryb pracy przelot
      AN    "Blok_Para".Wiazanie_Wzdluzne;
      AN    "Blok_Para".Wiazanie_Poprzeczne;
      =     "DB_HMI".HMI_IN.Wybrano_TP_Przelot;
//-wzdl
      A     "Blok_Para".Wiazanie_Wzdluzne;
      AN    "Blok_Para".Wiazanie_Poprzeczne;
      =     "DB_HMI".HMI_IN.Wybrano_TP_Wiazanie_Wzdl;
//-pop
      AN    "Blok_Para".Wiazanie_Wzdluzne;
      A     "Blok_Para".Wiazanie_Poprzeczne;
      =     "DB_HMI".HMI_IN.Wybrano_TP_Wiazanie_Pop;
//-pop -wzdl
      A     "Blok_Para".Wiazanie_Wzdluzne;
      A     "Blok_Para".Wiazanie_Poprzeczne;
      =     "DB_HMI".HMI_IN.Wybrano_TP_Wiazanie_Krzy;
NETWORK
TITLE =
//znacznik trybu wiazania
//krok_1  - przelot
      A     "DB_HMI".HMI_IN.Wybrano_TP_Przelot;
      L     1;
      JC    ztw;
//krok_2 - wzdluzna
      A     "DB_HMI".HMI_IN.Wybrano_TP_Wiazanie_Wzdl;
      L     2;
      JC    ztw;
//krok_3 - poprzeczne
      A     "DB_HMI".HMI_IN.Wybrano_TP_Wiazanie_Pop;
      L     3;
      JC    ztw;
//krok_4 - krzyzowe
      A     "DB_HMI".HMI_IN.Wybrano_TP_Wiazanie_Krzy;
      L     4;
      JC    ztw;
//daj 0
ztw:  T     "DB_HMI".HMI_IN.tryb_wiaz;
NETWORK
TITLE = Tryb Pracy Wiazanie wzduzne
//Zalaczenie Pozycjonowania
      A     "DB_HMI".HMI_IN_OUT.Tp_Pozycjonowanie;
      S     "Blok_Para".Pozycjonowanie;
      AN    "DB_HMI".HMI_IN_OUT.Tp_Pozycjonowanie;
      R     "Blok_Para".Pozycjonowanie;
      NOP   0;
NETWORK
TITLE = fotokomorka hamowania obrotnicy do kata 0st
//Fotokomorki katow pozycjonowania obrotnicy
      A     "AIO".Czuj_19_B.Czujnik_Ham_0_St;
      =     "DB_HMI".HMI_IN.Czujnik_Ham_0_St;
      A     "AIO".Czuj_19_B.Czujnik_0_St;
      =     "DB_HMI".HMI_IN.Czujnik_0_St;
      A     "AIO".Czuj_19_B.Czujnik_Ham_90_St;
      =     "DB_HMI".HMI_IN.Czujnik_Ham_90_St;
      A     "AIO".Czuj_19_B.Czujnik_90_St;
      =     "DB_HMI".HMI_IN.Czujnik_90_St;
      A     "AIO".Czuj_17_B.Czujnik_Ham_180_St;
      =     "DB_HMI".HMI_IN.Czujnik_Ham_180_St;
      A     "AIO".Czuj_17_B.Czujnik_180_St;
      =     "DB_HMI".HMI_IN.Czujnik_180_St;
      A     "AIO".Czuj_17_B.Czujnik_Ham_270_St;
      =     "DB_HMI".HMI_IN.Czujnik_Ham_270_St;
      A     "AIO".Czuj_17_B.Czujnik_270_St;
      =     "DB_HMI".HMI_IN.Czujnik_270_St;
NETWORK
TITLE = foto przednie bandzie wlotowej
//Fotokommorki
      A     "AIO".Banda_23.Foto_1;
      =     "DB_HMI".HMI_IN.Foto_Tasma_1_Przod;
      A     "AIO".Banda_23.Foto_2;
      =     "DB_HMI".HMI_IN.Foto_Tasma_1_Tyl;
      A     "AIO".Banda_24.Foto_1;
      =     "DB_HMI".HMI_IN.Foto_Tasma_2_Przod;
      A     "AIO".Banda_24.Foto_2;
      =     "DB_HMI".HMI_IN.Foto_Tasma_2_Tyl;
      A     "AIO".Obr_15.Foto_1;
      =     "DB_HMI".HMI_IN.Foto_Obrotnica_3_Przod;
      A     "AIO".Obr_15.Foto_2;
      =     "DB_HMI".HMI_IN.Foto_Obrotnica_3_Tyl;
      A     "AIO".Banda_2.Foto_1;
      =     "DB_HMI".HMI_IN.Foto_Tasma_4_Przod;
      A     "AIO".Banda_2.Foto_2;
      =     "DB_HMI".HMI_IN.Foto_Tasma_4_Tyl;
NETWORK
TITLE = tasma 1
//do wizualizacji przemieszczania palety na tasmie 1
      AN    "AIO".Banda_23.Foto_1;
      A     "AIO".Banda_23.Foto_2;
      =     "DB_HMI".HMI_IN.Paleta_na_Tasmie_1_T;
      A     "AIO".Banda_23.Foto_1;
      AN    "AIO".Banda_23.Foto_2;
      AN    "AIO".Banda_24.Foto_2;
      =     "DB_HMI".HMI_IN.Paleta_na_Tasmie_1_P;
      A     "AIO".Banda_23.Foto_1;
      A     "AIO".Banda_23.Foto_2;
      =     "DB_HMI".HMI_IN.Paleta_na_Tasmie_1;
NETWORK
TITLE = tasma 2
//do wizualizacji przemieszczania palety na tasmie 2
      AN    "AIO".Banda_24.Foto_1;
      A     "AIO".Banda_24.Foto_2;
      =     "DB_HMI".HMI_IN.Paleta_na_Tasmie_2_T;
      A     "AIO".Banda_24.Foto_1;
      AN    "AIO".Banda_24.Foto_2;
      AN    "AIO".Obr_15.Foto_1;
      =     "DB_HMI".HMI_IN.Paleta_na_Tasmie_2_P;
      A     "AIO".Banda_24.Foto_1;
      A     "AIO".Banda_24.Foto_2;
      =     "DB_HMI".HMI_IN.Paleta_na_Tasmie_2;
NETWORK
TITLE = tasma 3 (obrotnica)
//do wizualizacji przemieszczania palety na tasmie 3
      A     "AIO".Obr_15.Foto_1;
      AN    "AIO".Obr_15.Foto_2;
      A     "DB_HMI".HMI_IN.Czujnik_0_St;
      =     "DB_HMI".HMI_IN.Paleta_na_Tasmie_3_T;
      AN    "AIO".Obr_15.Foto_1;
      A     "AIO".Obr_15.Foto_2;
      AN    "AIO".Banda_2.Foto_2;
      A     "DB_HMI".HMI_IN.Czujnik_0_St;
      =     "DB_HMI".HMI_IN.Paleta_na_Tasmie_3_P;
      A     "AIO".Obr_15.Foto_1;
      A     "AIO".Obr_15.Foto_2;
      A(;
      O     "DB_HMI".HMI_IN.Czujnik_0_St;
      O     "DB_HMI".HMI_IN.Czujnik_180_St;
      );
      =     "DB_HMI".HMI_IN.Paleta_na_Tasmie_3_0_180;
      A     "AIO".Obr_15.Foto_1;
      A     "AIO".Obr_15.Foto_2;
      A(;
      O     "DB_HMI".HMI_IN.Czujnik_90_St;
      O     "DB_HMI".HMI_IN.Czujnik_270_St;
      );
      =     "DB_HMI".HMI_IN.Paleta_na_Tasmie_3_90_27;
NETWORK
TITLE = tasma 4
//do wizualizacji przemieszczania palety na tasmie 4
      AN    "AIO".Banda_2.Foto_1;
      A     "AIO".Banda_2.Foto_2;
      =     "DB_HMI".HMI_IN.Paleta_na_Tasmie_4_T;
      A     "AIO".Banda_2.Foto_1;
      AN    "AIO".Banda_2.Foto_2;
      =     "DB_HMI".HMI_IN.Paleta_na_Tasmie_4_P;
      A     "AIO".Banda_2.Foto_1;
      A     "AIO".Banda_2.Foto_2;
      =     "DB_HMI".HMI_IN.Paleta_na_Tasmie_4;
NETWORK
TITLE = motor obrotnica 3 counter clock wise
//Napedy band
      A     "AIO".Obr_15.CC_Wise;
      =     "DB_HMI".HMI_IN.Motor_Obrotnica_3_CCW;
      A     "AIO".Obr_15.C_Wise;
      =     "DB_HMI".HMI_IN.Motor_Obrotnica_3_CW;
      A     "AIO".Banda_23.CC_Wise;
      =     "DB_HMI".HMI_IN.Motor_Tasma_1_Przod;
      A     "AIO".Banda_23.C_Wise;
      =     "DB_HMI".HMI_IN.Motor_Tasma_1_Tyl;
      A     "AIO".Banda_24.C_Wise;
      =     "DB_HMI".HMI_IN.Motor_Tasma_2_Przod;
      A     "AIO".Banda_24.CC_Wise;
      =     "DB_HMI".HMI_IN.Motor_Tasma_2_Tyl;
      A     "AIO".Banda_1.C_Wise;
      =     "DB_HMI".HMI_IN.Motor_Tasma_3_Przod;
      A     "AIO".Banda_1.CC_Wise;
      =     "DB_HMI".HMI_IN.Motor_Tasma_3_Tyl;
      A     "AIO".Banda_2.CC_Wise;
      =     "DB_HMI".HMI_IN.Motor_Tasma_4_Przod;
      A     "AIO".Banda_2.C_Wise;
      =     "DB_HMI".HMI_IN.Motor_Tasma_4_Tyl;
NETWORK
TITLE = obwod bezpieczenstwa bindownicy
//sygnaly wymiany danych pomiedzy transportem palet a bindownica
      A     "Obwod_Bezp_Bindownicy";
      =     "DB_HMI".HMI_IN.Interfefs_B_do_TP_B1;
      A     "Bind_Polozenie_Podst";
      =     "DB_HMI".HMI_IN.Interfefs_B_do_TP_B2;
      A     "Start_Koniec_Wiazania";
      =     "DB_HMI".HMI_IN.Interfefs_B_do_TP_B3;
      A     "Bindownica_Auto";
      =     "DB_HMI".HMI_IN.Interfefs_B_do_TP_B4;
      A     "Blad_Bindownicy";
      =     "DB_HMI".HMI_IN.Interfefs_B_do_TP_B5;
//Transport do bindownicy 
      A     "Wirtualny_Sygnal_Bezp";
      =     "DB_HMI".HMI_IN.Interfefs_TP_do_B_TP1;
      A     "Zezw_na_prace_Bind";
      =     "DB_HMI".HMI_IN.Interfefs_TP_do_B_TP2;
      A     "o_Start_Wiazania";
      =     "DB_HMI".HMI_IN.Interfefs_TP_do_B_TP3;
NETWORK
TITLE = przycisk zalaczenie Strefy bezpieczenstwa
//przyciski, przelaczniki kierunkow i lampki na panelu
      A     "pb_Strefa_bezpieczenstwa";
      =     "DB_HMI".HMI_IN.PB_Strefa_bezpieczenstwa;
      A     "pb_Reczny";
      =     "DB_HMI".HMI_IN.PB_Reczny;
      A     "pb_Auto";
      =     "DB_HMI".HMI_IN.PB_Auto;
      A     "pb_Reset";
      =     "DB_HMI".HMI_IN.PB_Reset;
      A     "pb_Stop";
      =     "DB_HMI".HMI_IN.PB_Stop;
      A     "pb_Cykl_Start";
      =     "DB_HMI".HMI_IN.PB_Cykl_Start;
      A     "pb_Tasma_1_Tyl";
      =     "DB_HMI".HMI_IN.PB_Tasma1_Tyl;
      A     "pb_Tasma_1_Przod";
      =     "DB_HMI".HMI_IN.PB_Tasma1_Przod;
      A     "pb_Tasma_2_Tyl";
      =     "DB_HMI".HMI_IN.PB_Tasma2_Tyl;
      A     "pb_Tasma_2_Przod";
      =     "DB_HMI".HMI_IN.PB_Tasma2_Przod;
      A     "pb_Tasma_3_Tyl";
      =     "DB_HMI".HMI_IN.PB_Tasma3_Tyl;
      A     "pb_Tasma_3_Przod";
      =     "DB_HMI".HMI_IN.PB_Tasma3_Przod;
      A     "pb_Tasma_4_Tyl";
      =     "DB_HMI".HMI_IN.PB_Tasma4_Tyl;
      A     "pb_Tasma_4_Przod";
      =     "DB_HMI".HMI_IN.PB_Tasma4_Przod;
      A     "pb_Tasma_3_Obr_CW";
      =     "DB_HMI".HMI_IN.PB_Tasma3_Obr_CW;
      A     "pb_Tasma_3_Obr_CCW";
      =     "DB_HMI".HMI_IN.PB_Tasma3_Obr_CCW;
      A     "Lampka_Blad_Bind";
      =     "DB_HMI".HMI_IN.Lampka_Blad_Bind;
      A     "Lampka_Strzal_Tasmy";
      =     "DB_HMI".HMI_IN.Lampka_Strzal_Tasmy;
      A     "Lampka_pb_Strefa_Bezp";
      =     "DB_HMI".HMI_IN.Lampka_Strefa_Bezp;
      A     "Lampka_pb_Reczny";
      =     "DB_HMI".HMI_IN.Lampka_PB_Reczny;
      A     "Lampka_pb_Auto";
      =     "DB_HMI".HMI_IN.Lampka_PB_Auto;
      A     "Lampka_pb_Reset";
      =     "DB_HMI".HMI_IN.Lampka_PB_Reset;
      A     "Lampka_pb_Stop";
      =     "DB_HMI".HMI_IN.Lampka_PB_Stop;
      A     "Lampka_pb_Cykl_Start";
      =     "DB_HMI".HMI_IN.Lampka_PB_Cykl_Start;
NETWORK
TITLE =
//Start/Stop calej lini
      A     "DB_HMI".HMI_OUT.Start_Lini_z_OP;
      =     "Blok_Para".Start_Lini_z_OP;
      A     "DB_HMI".HMI_OUT.Stop_Lini_z_OP;
      =     "Blok_Para".Stop_Lini_z_OP;
NETWORK
TITLE = //wyjazd wtrybie auto
//Wyzwolenie wyjazdu palety gdy paleta stoi na bandzie obrotowej a nie wyjezdza
//
      A     "DB_HMI".HMI_OUT.Wyzwolenie_Wyjazdu;
      =     "Blok_Para".Trigger_Wyjazd;
NETWORK
TITLE = Znacznik stanu kurtyny optycznej na wlocie
//Bariery optyczne bindownicy
      AN    "AIO".Kurtyna_25.OSSD_Tor_1_1;
      AN    "AIO".Kurtyna_25.OSSD_Tor_1_2;
      AN    "AIO".Kurtyna_25.OSSD_Tor_2_1;
      AN    "AIO".Kurtyna_25.OSSD_Tor_2_2;
      =     "DB_HMI".HMI_IN.Kurtyna_Wlot_Ok;
      AN    "AIO".Kurtyna_26.OSSD_Tor_1_1;
      AN    "AIO".Kurtyna_26.OSSD_Tor_1_2;
      AN    "AIO".Kurtyna_26.OSSD_Tor_2_1;
      AN    "AIO".Kurtyna_26.OSSD_Tor_2_2;
      =     "DB_HMI".HMI_IN.Kurtyna_Wylot_Ok;
      A     "Rygiel_OK";
      =     "DB_HMI".HMI_IN.Rygiel;
NETWORK
TITLE = Znacznik pracy calej linii transportowej
      A     "Lampa_Zielona";
      =     "DB_HMI".HMI_IN.Linia_transportowa_praca;
NETWORK
TITLE = tryb pracy bindownicy: Auto(1) Reczny(0)
      A     "Blok_Bledow_Program".Blad_Krok_1;
      =     "DB_HMI".HMI_IN.Krok_1;
      A     "Blok_Bledow_Program".Blad_Krok_2;
      =     "DB_HMI".HMI_IN.Krok_2;
      A     "Blok_Bledow_Program".Blad_Krok_3;
      =     "DB_HMI".HMI_IN.Krok_3;
      A     "Blok_Bledow_Program".Blad_Krok_4;
      =     "DB_HMI".HMI_IN.Krok_4;
      A     "Blok_Bledow_Program".Blad_Krok_5;
      =     "DB_HMI".HMI_IN.Krok_5;
      A     "Blok_Bledow_Program".Blad_Krok_6;
      =     "DB_HMI".HMI_IN.Krok_6;
NETWORK
TITLE =
//przypisanie stanu wejsc i wyjsc
      L     "Bity_Przyciskow";
      T     "DB_HMI".HMI_IN.input_0;
      L     IB 1;
      T     "DB_HMI".HMI_IN.input_1;
      L     IB 2;
      T     "DB_HMI".HMI_IN.input_2;
      L     IB 3;
      T     "DB_HMI".HMI_IN.input_3;
      L     QB 0;
      T     "DB_HMI".HMI_IN.output_0;
      L     QB 1;
      T     "DB_HMI".HMI_IN.output_1;
      L     QB 2;
      T     "DB_HMI".HMI_IN.output_2;
      L     QB 3;
      T     "DB_HMI".HMI_IN.output_3;
      L     IB 8;
      T     "DB_HMI".HMI_IN.input_8;
      L     IB 9;
      T     "DB_HMI".HMI_IN.input_9;
      L     IB 10;
      T     "DB_HMI".HMI_IN.input_10;
      L     IB 11;
      T     "DB_HMI".HMI_IN.input_11;
NETWORK
TITLE = krok 1 trybu pracy
//Przypisanie aktualnych krokow 
//krok_1  - jedz na pozycje 
      A     "Blok_Para".Krok_1;
      L     1;
      JC    tr;
//krok_2 - szukaj srodka 
      A     "Blok_Para".krok_2;
      L     2;
      JC    tr;
//krok_3 - jedz na prawo
      A     "Blok_Para".krok_3;
      L     3;
      JC    tr;
//krok_4 - strzelaj 
      A     "Blok_Para".krok_4;
      L     4;
      JC    tr;
//krok_5  - pauza po strzale
      A     "Blok_Para".krok_5;
      L     5;
      JC    tr;
//krok_6 - jedz do srodka
      A     "Blok_Para".krok_6;
      L     6;
      JC    tr;
//daj 0
      L     0;
tr:   T     "DB_HMI".HMI_IN.INT_Liczba_Akt_Kroku;
NETWORK
TITLE = znacznik migania bledu
//Sprawdzenie czy sa bledy jak sa to miganie bledow
      SET;
      R     "DB_HMI".HMI_IN.Znacznik_Migania_Bledu;
      O(;
      L     DB119.DBD 0;
      L     0;
      <>D;
      );
      O(;
      L     DB119.DBD 4;
      L     0;
      <>D;
      );
      O(;
      L     DB119.DBD 8;
      L     0;
      <>D;
      );
      S     "DB_HMI".HMI_IN.Znacznik_Migania_Bledu;
NETWORK
TITLE = czujnik prasy s 22
//Obsluga wygladu prasy
//
      A     "Prasa_W_Gorze";
      =     "DB_HMI".HMI_IN.Czujnik_Prasa;
//zawor prasa
      AN    "Zawor_Prasa";
      =     "DB_HMI".HMI_IN.Stan_Zaworu;
NETWORK
TITLE =
//Aktualizacja godziny/daty panela z godzina/czasem PLC
      CALL  "READ_CLK" (
           RET_VAL                  := #LW0_Help,
           CDT                      := "DB_HMI".HMI_IN.Aktualna_Data);
END_FUNCTION

FUNCTION "Funkcja_Zegara" : VOID	// FC 140
AUTHOR : Kng
NAME : HELP_FC
VERSION : 0.1
VAR_INPUT
  Timer_NR : TIMER ;
  Czas : S5TIME ;
END_VAR
VAR_IN_OUT
  Wyjscie : BOOL ;
END_VAR
BEGIN
NETWORK
TITLE =
      A     #Timer_NR;
      SAVE;
      NOT;
      L     #Czas;
      SD    #Timer_NR;
      X     BR;
      X     #Wyjscie;
      =     #Wyjscie;
END_FUNCTION

DATA_BLOCK DB 2
VERSION : 0.0
"TEST_OBR2"
BEGIN
END_DATA_BLOCK

DATA_BLOCK DB 4
VERSION : 0.0
"Czesc_Bindujaca"
BEGIN
END_DATA_BLOCK

DATA_BLOCK DB 5
VERSION : 0.0
"Blok_Jazdy_Band"
BEGIN
END_DATA_BLOCK

DATA_BLOCK "AIO"	// DB 10
VERSION : 0.1
  STRUCT
   Banda_1 : UDT 1;	//Temporary placeholder variable
   Banda_2 : UDT 1;
   Banda_3 : UDT 1;
   Banda_4 : UDT 9;
   Banda_5 : UDT 1;
   Banda_6 : UDT 1;
   Banda_7 : UDT 1;
   Banda_8 : UDT 1;
   Banda_9 : UDT 1;
   Banda_10 : UDT 1;
   Banda_11 : UDT 1;
   Banda_12 : UDT 1;
   Banda_13 : UDT 9;
   Banda_14 : UDT 1;
   Obr_15 : UDT 11;
   Czuj_19_B : UDT 7;
   Czuj_17_B : UDT 10;
   Obr_18 : UDT 6;
   Czuj_19 : UDT 7;
   Obr_20 : UDT 6;
   Czuj_21 : UDT 7;
   Czuj_22 : UDT 8;
   Banda_23 : UDT 1;
   Banda_24 : UDT 1;
   Kurtyna_25 : UDT 2;
   Kurtyna_26 : UDT 2;
   ESTOP_27 : UDT 3;
   ESTOP_28 : UDT 3;
   ESTOP_29 : UDT 3;
   ESTOP_30 : UDT 3;
   ESTOP_31 : UDT 3;
   Rygiel_16 : UDT 2;
   Reset_17 : UDT 12;
  END_STRUCT ;	
BEGIN
END_DATA_BLOCK

DATA_BLOCK DB 11
VERSION : 0.0
FB 1
BEGIN
END_DATA_BLOCK

DATA_BLOCK "Blok_Para"	// DB 12
VERSION : 0.1
  STRUCT
   Wiazanie_Poprzeczne : BOOL ;	//Wiaz wzdluz
   Wiazanie_Wzdluzne : BOOL ;
   Pozycjonowanie : BOOL ;
   Przelacz_Na_Auto : BOOL ;	//warunkowe przejscie na auto
   Start_Lini_z_OP : BOOL ;
   Stop_Lini_z_OP : BOOL ;
   Trigger_Wyjazd : BOOL ;	////wyjazd wtrybie auto
   Ser_Pokrycie_Foto : BOOL ;
   Pozycjon_Banda_Lewo : BOOL ;
   Pozycjon_Banda_Prawo : BOOL ;
   Pozycjon_Banda_Srodek : BOOL ;	//rozakaz pozycjonowana
   Banda_Poz_Lewa : BOOL ;
   Banda_Poz_Prawa : BOOL ;
   Banda_Poz_Srodek : BOOL ;
   Banda_Poz_Potw : BOOL ;
   Jedz_Na_0st : BOOL ;
   Jedz_Na_90st : BOOL ;
   Jedz_Na_180st : BOOL ;
   Jedz_Na_270st : BOOL ;
   Poz_0_st : BOOL ;
   Poz_90_st : BOOL ;
   Poz_180_st : BOOL ;
   Poz_270_st : BOOL ;
   Poz_Obr_Osiagnieta : BOOL ;
   Odblokuj_Rolki : BOOL ;
   Odblokuj_Obrotnice : BOOL ;
   Poz_Obr_Osiagnieta1 : BOOL ;
   Pozycja_Obrotnicy : INT ;
   Bin_Licznik : INT ;	//licznik bindownicy
   Rezerwa_Para : DWORD ;
   Krok_1 : BOOL ;
   krok_2 : BOOL ;
   krok_3 : BOOL ;
   krok_4 : BOOL ;
   krok_5 : BOOL ;
   krok_6 : BOOL ;
   krok_7 : BOOL ;
   krok_8 : BOOL ;
   krok_9 : BOOL ;
  END_STRUCT ;	
BEGIN
END_DATA_BLOCK

DATA_BLOCK "Blok_Bledow_Program"	// DB 13
VERSION : 0.1
  STRUCT
   Blad_Krok_1 : BOOL ;	//Blad kroku nr 1 (Przekrokczony czas jazdy  na zadana pozycje)
   Blad_Krok_2 : BOOL ;	//Blad kroku nr 2 (Przekrokczony czas szukania srodka palety)
   Blad_Krok_3 : BOOL ;	//Blad kroku nr 3 (Przekrokczony czas pozycjonowania palety lewo/prawo)
   Blad_Krok_4 : BOOL ;	//Blad kroku nr 4 (Przekrokczony czas strzalu bindownicy)
   Blad_Krok_5 : BOOL ;	//Blad kroku nr 6 (Przekrokczony czas czasu postoju)
   Blad_Krok_6 : BOOL ;	//Blad kroku nr 5 (Przekrokczony czas powrotu lewo/prawo)
   Blad_Krok_7 : BOOL ;	//Rezerwa
   Blad_Krok_8 : BOOL ;	//Rezerwa
   Blad_Krok_9 : BOOL ;	//Rezerwa
   Blad_Krok_10 : BOOL ;	//Rezerwa
  END_STRUCT ;	
BEGIN
END_DATA_BLOCK

DATA_BLOCK DB 20
AUTHOR : Kng
VERSION : 0.0
"T_ON"
BEGIN
END_DATA_BLOCK

DATA_BLOCK DB 33
VERSION : 0.0
FB 1
BEGIN
END_DATA_BLOCK

DATA_BLOCK "Asi_input"	// DB 80
VERSION : 0.1
  STRUCT
   Adres_1_bit_0 : BOOL ;	//Temporary placeholder variable
   Adres_1_bit_1 : BOOL ;
   Adres_1_bit_2 : BOOL ;
   Adres_1_bit_3 : BOOL ;
   Adres_0_bit_0 : BOOL ;	//Temporary placeholder variable
   Adres_0_bit_1 : BOOL ;
   Adres_0_bit_2 : BOOL ;
   Adres_0_bit_3 : BOOL ;
   Adres_3_bit_0 : BOOL ;	//Temporary placeholder variable
   Adres_3_bit_1 : BOOL ;
   Adres_3_bit_2 : BOOL ;
   Adres_3_bit_3 : BOOL ;
   Adres_2_bit_0 : BOOL ;	//Temporary placeholder variable
   Adres_2_bit_1 : BOOL ;
   Adres_2_bit_2 : BOOL ;
   Adres_2_bit_3 : BOOL ;
   Adres_5_bit_0 : BOOL ;	//Temporary placeholder variable
   Adres_5_bit_1 : BOOL ;
   Adres_5_bit_2 : BOOL ;
   Adres_5_bit_3 : BOOL ;
   Adres_4_bit_0 : BOOL ;	//Temporary placeholder variable
   Adres_4_bit_1 : BOOL ;
   Adres_4_bit_2 : BOOL ;
   Adres_4_bit_3 : BOOL ;
   Adres_7_bit_0 : BOOL ;	//Temporary placeholder variable
   Adres_7_bit_1 : BOOL ;
   Adres_7_bit_2 : BOOL ;
   Adres_7_bit_3 : BOOL ;
   Adres_6_bit_0 : BOOL ;	//Temporary placeholder variable
   Adres_6_bit_1 : BOOL ;
   Adres_6_bit_2 : BOOL ;
   Adres_6_bit_3 : BOOL ;
   Adres_9_bit_0 : BOOL ;	//Temporary placeholder variable
   Adres_9_bit_1 : BOOL ;
   Adres_9_bit_2 : BOOL ;
   Adres_9_bit_3 : BOOL ;
   Adres_8_bit_0 : BOOL ;	//Temporary placeholder variable
   Adres_8_bit_1 : BOOL ;
   Adres_8_bit_2 : BOOL ;
   Adres_8_bit_3 : BOOL ;
   Adres_11_bit_0 : BOOL ;	//Temporary placeholder variable
   Adres_11_bit_1 : BOOL ;
   Adres_11_bit_2 : BOOL ;
   Adres_11_bit_3 : BOOL ;
   Adres_10_bit_0 : BOOL ;	//Temporary placeholder variable
   Adres_10_bit_1 : BOOL ;
   Adres_10_bit_2 : BOOL ;
   Adres_10_bit_3 : BOOL ;
   Adres_13_bit_0 : BOOL ;	//Temporary placeholder variable
   Adres_13_bit_1 : BOOL ;
   Adres_13_bit_2 : BOOL ;
   Adres_13_bit_3 : BOOL ;
   Adres_12_bit_0 : BOOL ;	//Temporary placeholder variable
   Adres_12_bit_1 : BOOL ;
   Adres_12_bit_2 : BOOL ;
   Adres_12_bit_3 : BOOL ;
   Adres_15_bit_0 : BOOL ;	//Temporary placeholder variable
   Adres_15_bit_1 : BOOL ;
   Adres_15_bit_2 : BOOL ;
   Adres_15_bit_3 : BOOL ;
   Adres_14_bit_0 : BOOL ;	//Temporary placeholder variable
   Adres_14_bit_1 : BOOL ;
   Adres_14_bit_2 : BOOL ;
   Adres_14_bit_3 : BOOL ;
   Adres_17_bit_0 : BOOL ;	//Temporary placeholder variable
   Adres_17_bit_1 : BOOL ;
   Adres_17_bit_2 : BOOL ;
   Adres_17_bit_3 : BOOL ;
   Adres_16_bit_0 : BOOL ;	//Temporary placeholder variable
   Adres_16_bit_1 : BOOL ;
   Adres_16_bit_2 : BOOL ;
   Adres_16_bit_3 : BOOL ;
   Adres_19_bit_0 : BOOL ;	//Temporary placeholder variable
   Adres_19_bit_1 : BOOL ;
   Adres_19_bit_2 : BOOL ;
   Adres_19_bit_3 : BOOL ;
   Adres_18_bit_0 : BOOL ;	//Temporary placeholder variable
   Adres_18_bit_1 : BOOL ;
   Adres_18_bit_2 : BOOL ;
   Adres_18_bit_3 : BOOL ;
   Adres_21_bit_0 : BOOL ;	//Temporary placeholder variable
   Adres_21_bit_1 : BOOL ;
   Adres_21_bit_2 : BOOL ;
   Adres_21_bit_3 : BOOL ;
   Adres_20_bit_0 : BOOL ;	//Temporary placeholder variable
   Adres_20_bit_1 : BOOL ;
   Adres_20_bit_2 : BOOL ;
   Adres_20_bit_3 : BOOL ;
   Adres_23_bit_0 : BOOL ;	//Temporary placeholder variable
   Adres_23_bit_1 : BOOL ;
   Adres_23_bit_2 : BOOL ;
   Adres_23_bit_3 : BOOL ;
   Adres_22_bit_0 : BOOL ;	//Temporary placeholder variable
   Adres_22_bit_1 : BOOL ;
   Adres_22_bit_2 : BOOL ;
   Adres_22_bit_3 : BOOL ;
   Adres_25_bit_0 : BOOL ;	//Temporary placeholder variable
   Adres_25_bit_1 : BOOL ;
   Adres_25_bit_2 : BOOL ;
   Adres_25_bit_3 : BOOL ;
   Adres_24_bit_0 : BOOL ;	//Temporary placeholder variable
   Adres_24_bit_1 : BOOL ;
   Adres_24_bit_2 : BOOL ;
   Adres_24_bit_3 : BOOL ;
   Adres_27_bit_0 : BOOL ;	//Temporary placeholder variable
   Adres_27_bit_1 : BOOL ;
   Adres_27_bit_2 : BOOL ;
   Adres_27_bit_3 : BOOL ;
   Adres_26_bit_0 : BOOL ;	//Temporary placeholder variable
   Adres_26_bit_1 : BOOL ;
   Adres_26_bit_2 : BOOL ;
   Adres_26_bit_3 : BOOL ;
   Adres_29_bit_0 : BOOL ;	//Temporary placeholder variable
   Adres_29_bit_1 : BOOL ;
   Adres_29_bit_2 : BOOL ;
   Adres_29_bit_3 : BOOL ;
   Adres_28_bit_0 : BOOL ;	//Temporary placeholder variable
   Adres_28_bit_1 : BOOL ;
   Adres_28_bit_2 : BOOL ;
   Adres_28_bit_3 : BOOL ;
   Adres_31_bit_0 : BOOL ;	//Temporary placeholder variable
   Adres_31_bit_1 : BOOL ;
   Adres_31_bit_2 : BOOL ;
   Adres_31_bit_3 : BOOL ;
   Adres_30_bit_0 : BOOL ;	//Temporary placeholder variable
   Adres_30_bit_1 : BOOL ;
   Adres_30_bit_2 : BOOL ;
   Adres_30_bit_3 : BOOL ;
   B_Adres_1_bit_0 : BOOL ;	//Temporary placeholder variable
   B_Adres_1_bit_1 : BOOL ;
   B_Adres_1_bit_2 : BOOL ;
   B_Adres_1_bit_3 : BOOL ;
   B_Adres_0_bit_0 : BOOL ;
   B_Adres_0_bit_1 : BOOL ;
   B_Adres_0_bit_2 : BOOL ;
   B_Adres_0_bit_3 : BOOL ;
   B_Adres_3_bit_0 : BOOL ;	//Temporary placeholder variable
   B_Adres_3_bit_1 : BOOL ;
   B_Adres_3_bit_2 : BOOL ;
   B_Adres_3_bit_3 : BOOL ;
   B_Adres_2_bit_0 : BOOL ;	//Temporary placeholder variable
   B_Adres_2_bit_1 : BOOL ;
   B_Adres_2_bit_2 : BOOL ;
   B_Adres_2_bit_3 : BOOL ;
   B_Adres_5_bit_0 : BOOL ;	//Temporary placeholder variable
   B_Adres_5_bit_1 : BOOL ;
   B_Adres_5_bit_2 : BOOL ;
   B_Adres_5_bit_3 : BOOL ;
   B_Adres_4_bit_0 : BOOL ;	//Temporary placeholder variable
   B_Adres_4_bit_1 : BOOL ;
   B_Adres_4_bit_2 : BOOL ;
   B_Adres_4_bit_3 : BOOL ;
   B_Adres_7_bit_0 : BOOL ;	//Temporary placeholder variable
   B_Adres_7_bit_1 : BOOL ;
   B_Adres_7_bit_2 : BOOL ;
   B_Adres_7_bit_3 : BOOL ;
   B_Adres_6_bit_0 : BOOL ;	//Temporary placeholder variable
   B_Adres_6_bit_1 : BOOL ;
   B_Adres_6_bit_2 : BOOL ;
   B_Adres_6_bit_3 : BOOL ;
   B_Adres_9_bit_0 : BOOL ;	//Temporary placeholder variable
   B_Adres_9_bit_1 : BOOL ;
   B_Adres_9_bit_2 : BOOL ;
   B_Adres_9_bit_3 : BOOL ;
   B_Adres_8_bit_0 : BOOL ;	//Temporary placeholder variable
   B_Adres_8_bit_1 : BOOL ;
   B_Adres_8_bit_2 : BOOL ;
   B_Adres_8_bit_3 : BOOL ;
   B_Adres_11_bit_0 : BOOL ;	//Temporary placeholder variable
   B_Adres_11_bit_1 : BOOL ;
   B_Adres_11_bit_2 : BOOL ;
   B_Adres_11_bit_3 : BOOL ;
   B_Adres_10_bit_0 : BOOL ;	//Temporary placeholder variable
   B_Adres_10_bit_1 : BOOL ;
   B_Adres_10_bit_2 : BOOL ;
   B_Adres_10_bit_3 : BOOL ;
   B_Adres_13_bit_0 : BOOL ;	//Temporary placeholder variable
   B_Adres_13_bit_1 : BOOL ;
   B_Adres_13_bit_2 : BOOL ;
   B_Adres_13_bit_3 : BOOL ;
   B_Adres_12_bit_0 : BOOL ;	//Temporary placeholder variable
   B_Adres_12_bit_1 : BOOL ;
   B_Adres_12_bit_2 : BOOL ;
   B_Adres_12_bit_3 : BOOL ;
   B_Adres_15_bit_0 : BOOL ;	//Temporary placeholder variable
   B_Adres_15_bit_1 : BOOL ;
   B_Adres_15_bit_2 : BOOL ;
   B_Adres_15_bit_3 : BOOL ;
   B_Adres_14_bit_0 : BOOL ;	//Temporary placeholder variable
   B_Adres_14_bit_1 : BOOL ;
   B_Adres_14_bit_2 : BOOL ;
   B_Adres_14_bit_3 : BOOL ;
   B_Adres_17_bit_0 : BOOL ;	//Temporary placeholder variable
   B_Adres_17_bit_1 : BOOL ;
   B_Adres_17_bit_2 : BOOL ;
   B_Adres_17_bit_3 : BOOL ;
   B_Adres_16_bit_0 : BOOL ;	//Temporary placeholder variable
   B_Adres_16_bit_1 : BOOL ;
   B_Adres_16_bit_2 : BOOL ;
   B_Adres_16_bit_3 : BOOL ;
   B_Adres_19_bit_0 : BOOL ;	//Temporary placeholder variable
   B_Adres_19_bit_1 : BOOL ;
   B_Adres_19_bit_2 : BOOL ;
   B_Adres_19_bit_3 : BOOL ;
   B_Adres_18_bit_0 : BOOL ;	//Temporary placeholder variable
   B_Adres_18_bit_1 : BOOL ;
   B_Adres_18_bit_2 : BOOL ;
   B_Adres_18_bit_3 : BOOL ;
   B_Adres_21_bit_0 : BOOL ;	//Temporary placeholder variable
   B_Adres_21_bit_1 : BOOL ;
   B_Adres_21_bit_2 : BOOL ;
   B_Adres_21_bit_3 : BOOL ;
   B_Adres_20_bit_0 : BOOL ;	//Temporary placeholder variable
   B_Adres_20_bit_1 : BOOL ;
   B_Adres_20_bit_2 : BOOL ;
   B_Adres_20_bit_3 : BOOL ;
   B_Adres_23_bit_0 : BOOL ;	//Temporary placeholder variable
   B_Adres_23_bit_1 : BOOL ;
   B_Adres_23_bit_2 : BOOL ;
   B_Adres_23_bit_3 : BOOL ;
   B_Adres_22_bit_0 : BOOL ;	//Temporary placeholder variable
   B_Adres_22_bit_1 : BOOL ;
   B_Adres_22_bit_2 : BOOL ;
   B_Adres_22_bit_3 : BOOL ;
   B_Adres_25_bit_0 : BOOL ;	//Temporary placeholder variable
   B_Adres_25_bit_1 : BOOL ;
   B_Adres_25_bit_2 : BOOL ;
   B_Adres_25_bit_3 : BOOL ;
   B_Adres_24_bit_0 : BOOL ;	//Temporary placeholder variable
   B_Adres_24_bit_1 : BOOL ;
   B_Adres_24_bit_2 : BOOL ;
   B_Adres_24_bit_3 : BOOL ;
   B_Adres_27_bit_0 : BOOL ;	//Temporary placeholder variable
   B_Adres_27_bit_1 : BOOL ;
   B_Adres_27_bit_2 : BOOL ;
   B_Adres_27_bit_3 : BOOL ;
   B_Adres_26_bit_0 : BOOL ;	//Temporary placeholder variable
   B_Adres_26_bit_1 : BOOL ;
   B_Adres_26_bit_2 : BOOL ;
   B_Adres_26_bit_3 : BOOL ;
   B_Adres_29_bit_0 : BOOL ;	//Temporary placeholder variable
   B_Adres_29_bit_1 : BOOL ;
   B_Adres_29_bit_2 : BOOL ;
   B_Adres_29_bit_3 : BOOL ;
   B_Adres_28_bit_0 : BOOL ;	//Temporary placeholder variable
   B_Adres_28_bit_1 : BOOL ;
   B_Adres_28_bit_2 : BOOL ;
   B_Adres_28_bit_3 : BOOL ;
   B_Adres_31_bit_0 : BOOL ;	//Temporary placeholder variable
   B_Adres_31_bit_1 : BOOL ;
   B_Adres_31_bit_2 : BOOL ;
   B_Adres_31_bit_3 : BOOL ;
   B_Adres_30_bit_0 : BOOL ;	//Temporary placeholder variable
   B_Adres_30_bit_1 : BOOL ;
   B_Adres_30_bit_2 : BOOL ;
   B_Adres_30_bit_3 : BOOL ;
  END_STRUCT ;	
BEGIN
END_DATA_BLOCK

